                   #S120_SHUTTLE_TO_EXT_LOAD_UNLOAD_POS_START_REQ:
                       REGION S120_SHUTTLE_TO_EXT_LOAD_UNLOAD_POS_START_REQ
                           IF #sInterface.SequenceReleased AND #sStepForward AND (#iShuttleMoving OR #iShuttleModeSemiAutoPos) THEN
                               #sCurrent_Step_NB := #S130_SHUTTLE_TO_EXT_LOAD_UNLOAD_POS_REACHED;
                               #sCheck_Step_Condition := FALSE;
                           END_IF;
                       END_REGION
                   #S130_SHUTTLE_TO_EXT_LOAD_UNLOAD_POS_REACHED:
                       REGION S130_SHUTTLE_TO_EXT_LOAD_UNLOAD_POS_REACHED
                           IF #sInterface.SequenceReleased AND #sStepForward AND NOT #sShuttleStartReq AND #iShuttleModeSemiAutoPos THEN
                               #sCurrent_Step_NB := #S140_STOP_CYCLE;
                               #sCheck_Step_Condition := FALSE;
                           END_IF;
                       END_REGION
                   #S140_STOP_CYCLE:
                       REGION S140_STOP_CYCLE
                           IF #sInterface.SequenceReleased AND #sStepForward AND #iNC_Stopped THEN
                               #sCurrent_Step_NB := #S150_WAIT_OPERATOR_RESTART;
                               #sCheck_Step_Condition := FALSE;
                           END_IF;
                       END_REGION
                       #S150_WAIT_OPERATOR_RESTART:
                           REGION S150_EXCHANGE_EXT_LOADER_IN_PROGRESS
                               IF #sInterface.SequenceReleased AND #sStepForward AND #iOperatorCycleRestart THEN
                                   #sCurrent_Step_NB := #S160_NC_RESTART;
                                   #sCheck_Step_Condition := FALSE;
                               END_IF;
                           END_REGION
                       #S160_NC_RESTART:
                           REGION S60_NC_RESTART
                               IF #sInterface.SequenceReleased AND #sStepForward AND #iNC_Running THEN
                                   #sCurrent_Step_NB := #S170_UPDATE_NEXT_STEP;
                                   #sCheck_Step_Condition := FALSE;
                               END_IF;
                           END_REGION
                       #S170_UPDATE_NEXT_STEP:
                           REGION S70_UPDATE_NEXT_STEP
                               IF #sInterface.SequenceReleased AND #sStepForward AND "AlwaysTRUE" THEN
                                   #sCurrent_Step_NB := #S295_JOB_DONE;
                                   #sCheck_Step_Condition := FALSE;
                               END_IF;
                           END_REGION
                       #S270_UPDATE_NEXT_STEP:
                           REGION S270_UPDATE_NEXT_STEP
                               IF #sInterface.SequenceReleased AND #sStepForward AND "AlwaysTRUE" THEN
                                   #sCurrent_Step_NB := #S295_JOB_DONE;
                                   #sCheck_Step_Condition := FALSE;
                               END_IF;
                           END_REGION
                       #S295_JOB_DONE:
                           REGION S295_JOB_DONE
                               IF NOT #iJobReq THEN
                                   #sCurrent_Step_NB := #S00_INIT;
                                   #sCheck_Step_Condition := FALSE;
                                   #sInterface.JobDone := FALSE;
                               END_IF;
                           END_REGION
               ELSE
                   #sInterface.Error := TRUE;
           END_CASE;
       END_IF;
   END_REGION

   REGION Outputs Update
       #oShuttleStartReq := #sShuttleStartReq;
       #oShuttlePosSetPoint := #sShuttlePosSetPoint;
       #oStopNC_Req := #sStopNC_Req;
       #oRestartNC_Req := #sRestartNC_Req;
       #oRestartStep := #sRestartStep;
       #oContinuationStep := #sContinuationStep;
       #oMsgMissingPart := #sMsgMissingPart;
       #oMsgExtraPart := #sMsgExtraPart;
   END_REGION

   REGION Steps - Date and Time History
       IF #sHistory.Activation THEN
           IF #sHistory.Steps[0] <> #sCurrent_Step_NB THEN
               FOR #tIndex := 98 TO 0 BY -1 DO
                   #sHistory.Steps[#tIndex + 1] := #sHistory.Steps[#tIndex];
                   #sHistory.Date_Time[#tIndex + 1] := #sHistory.Date_Time[#tIndex];
               END_FOR;
               #sHistory.Steps[0] := #sCurrent_Step_NB;
               #sHistory.Date_Time[0] := #iPLC_DateAndTime;
           END_IF;
       END_IF;
   END_REGION

   REGION Steps Text
       #StepText(iErrorCode := #sCurrent_Step_NB,
                 oErrorText => #StepText.oErrorText);
   END_REGION
END_FUNCTION_BLOCK

FUNCTION_BLOCK "FB_LoaderShuttle2"   // FB205, SCL
{ S7_Optimized_Access := 'TRUE' }
// stored: AutoNumber false, MemoryReserve 100, SetENOAutomatically false
   VAR_INPUT
      iGripperReserved : Bool;
      iGripperReleased : Bool;
      iShuttleMoving : Bool;
      iShuttleInPos : Bool;
      iAxisV_Moving : Bool;
      iAxisV_InPos : Bool;
      iAxisW_Moving : Bool;
      iAxisW_InPos : Bool;
   END_VAR
   VAR_OUTPUT
      oExtGateOpenReq : Bool;
      oExtGateCloseReq : Bool;
      oIntGateOpenReq : Bool;
      oIntGateCloseReq : Bool;
      oLoadGripperCloseReq : Bool;
      oUnloadGripperOpenReq : Bool;
      oBlowingReq : Bool;
      oShuttleStartReq : Bool;
      oShuttlePosSetPoint : Real;
      oAxisVStartReq : Bool;
      oAxisVPosSetPoint : Real;
      oAxisWStartReq : Bool;
      oAxisWPosSetPoint : Real;
   END_VAR
   VAR
      sMain : "FB_Main";
      sShuttleInt { S7_SetPoint := 'True'} : "FB_ShuttleInt";
      sShuttleExt { S7_SetPoint := 'True'} : "FB_ShuttleExt";
      sControlIn { S7_SetPoint := 'True'} : "FB_PartControl";
      sControlOut { S7_SetPoint := 'True'} : "FB_PartControl";
      sBlowing { S7_SetPoint := 'True'} : "FB_Blowing";
      sIntLoadUnload { S7_SetPoint := 'True'} : "FB_IntLoadUnload";
      sExtLoadUnload { S7_SetPoint := 'True'} : "FB_ExtLoadUnload";
      sBwLoadUnload { S7_SetPoint := 'True'} : "FB_BwLoadUnload";
      sBwControlIn { S7_SetPoint := 'True'} : "FB_BwControl";
      sActPartControlIn { S7_SetPoint := 'True'} : "FB_ActControl";
      sActPartControlout { S7_SetPoint := 'True'} : "FB_ActControl";
      sActBwControlIn { S7_SetPoint := 'True'} : "FB_ActControl";
      sIntLoadUnloadOP { S7_SetPoint := 'True'} : "FB_IntLoadUnloadOP";
      sBwConsecutiveCtrl_1 { S7_SetPoint := 'True'} : "FB_Consecutive";
      sBwConsecutiveCtrl { S7_SetPoint := 'True'} : "FB_Consecutive";
      sShuttlePosInt { S7_SetPoint := 'True'} : Bool;
      sShuttlePosSas : Bool;
      sShuttlePosExt : Bool;
      sGripper_OK : Bool;
      sExtLoaderInSafePos : Bool;
      sIntLoaderInSafePos : Bool;
      sBwLoaderInSafePos : Bool;
      sRT_PartControlInMissing : R_TRIG;
      sRT_PartControlInExtra : R_TRIG;
      sRT_PartControlOutMissing : R_TRIG;
      sRT_PartControlOutExtra : R_TRIG;
      sRT_BwControlInMissing : R_TRIG;
      sRT_BwControlInExtra : R_TRIG;
      sStepPauseSeq { S7_SetPoint := 'True'} : Bool;
   END_VAR
   VAR_TEMP
      tAxis_U_Position : Struct
         ExtLoadUnloadAuto : Bool;
         ExtLoadUnloadManu : Bool;
         PartControl : Bool;
         BwLoad : Bool;
         BwUnload : Bool;
         BwControl : Bool;
         IntLoadUnload : Bool;
         Blowing : Bool;
         IntLoadUnloadOP : Bool;
      END_STRUCT;
      tAxis_V_Position : Struct
         LoadUnload : Bool;
         Safe : Bool;
         Blowing : Bool;
      END_STRUCT;
      tAxis_W_Position : Struct
         LoadUnload : Bool;
         Safe : Bool;
         Approach : Bool;
         Blowing : Bool;
      END_STRUCT;
   END_VAR
BEGIN
   REGION Shuttle 2 position
       // Init Position
       #sShuttlePosInt := FALSE;
       #sShuttlePosSas := FALSE;
       #sShuttlePosExt := FALSE;

       // Check Shuttle (U2 Axis) position
       IF "DB_AxisPosition".sAxis06_U2."$AA_IM" < "DB_AxisPosMachinePLC".Axis_U2.IntGateExt THEN
           #sShuttlePosExt := TRUE;
       ELSIF "DB_AxisPosition".sAxis06_U2."$AA_IM" > "DB_AxisPosMachinePLC".Axis_U2.ExtGateInt THEN
           #sShuttlePosInt := TRUE;
       ELSE
           #sShuttlePosSas := TRUE;
       END_IF;
   END_REGION

   REGION Position Check
       REGION Axis U2
           // Position : External Load / Unload Auto
           "FC_PositionCheck"(iAxisCurrentPos := "DB_AxisPosition".sAxis06_U2."$AA_IM",
                              iAxisTargetPos := "DB_AxisPosMachinePLC".Axis_U2.ExtLoadUnloadAuto,
                              iTolMin := 0.001,
                              iTolMax := 0.001,
                              iInPos => #tAxis_U_Position.ExtLoadUnloadAuto);

           // Position : External Load / Unload Manu
           "FC_PositionCheck"(iAxisCurrentPos := "DB_AxisPosition".sAxis06_U2."$AA_IM",
                              iAxisTargetPos := "DB_AxisPosMachinePLC".Axis_U2.ExtLoadUnloadManu,
                              iTolMin := 0.001,
                              iTolMax := 0.001,
                              iInPos => #tAxis_U_Position.ExtLoadUnloadManu);

           // Position : Part Control
           "FC_PositionCheck"(iAxisCurrentPos := "DB_AxisPosition".sAxis06_U2."$AA_IM",
                              iAxisTargetPos := "DB_AxisPosMachinePLC".Axis_U2.PartControl,
                              iTolMin := 0.001,
                              iTolMax := 0.001,
                              iInPos => #tAxis_U_Position.PartControl);

           // Position : Backwall Load
           "FC_PositionCheck"(iAxisCurrentPos := "DB_AxisPosition".sAxis06_U2."$AA_IM",
                              iAxisTargetPos := "DB_AxisPosMachinePLC".Axis_U2.BwLoad,
                              iTolMin := 0.001,
                              iTolMax := 0.001,
                              iInPos => #tAxis_U_Position.BwLoad);

           // Position : Backwall Unload
           "FC_PositionCheck"(iAxisCurrentPos := "DB_AxisPosition".sAxis06_U2."$AA_IM",
                              iAxisTargetPos := "DB_AxisPosMachinePLC".Axis_U2.BwUnLoad,
                              iTolMin := 0.001,
                              iTolMax := 0.001,
                              iInPos => #tAxis_U_Position.BwUnload);

           // Position : Backwall Control
           "FC_PositionCheck"(iAxisCurrentPos := "DB_AxisPosition".sAxis06_U2."$AA_IM",
                              iAxisTargetPos := "DB_AxisPosMachinePLC".Axis_U2.BwControl,
                              iTolMin := 0.001,
                              iTolMax := 0.001,
                              iInPos => #tAxis_U_Position.BwControl);

           // Position : Internal Load / Unload
           "FC_PositionCheck"(iAxisCurrentPos := "DB_AxisPosition".sAxis06_U2."$AA_IM",
                              iAxisTargetPos := "DB_AxisPosMachinePLC".Axis_U2.IntLoadUnload,
                              iTolMin := 0.001,
                              iTolMax := 0.001,
                              iInPos => #tAxis_U_Position.IntLoadUnload);

           // Position : Internal Load / Unload OP
           "FC_PositionCheck"(iAxisCurrentPos := "DB_AxisPosition".sAxis06_U2."$AA_IM",
                              iAxisTargetPos := "DB_AxisPosMachinePLC".Axis_U2.IntLoadUnloadOP,
                              iTolMin := 0.001,
                              iTolMax := 0.001,
                              iInPos => #tAxis_U_Position.IntLoadUnloadOP);

           // Position : Blowing (Undrilled part)
           "FC_PositionCheck"(iAxisCurrentPos := "DB_AxisPosition".sAxis06_U2."$AA_IM",
                              iAxisTargetPos := "DB_AxisPosMachinePLC".Axis_U2.Blowing,
                              iTolMin := 0.001,
                              iTolMax := 0.001,
                              iInPos => #tAxis_U_Position.Blowing);
       END_REGION

       REGION Axis V
           // Position : Load / Unload Auto
           "FC_PositionCheck"(iAxisCurrentPos := "DB_AxisPosition".sAxis07_V."$AA_IM",
                              iAxisTargetPos := "DB_AxisPosMachinePLC".Axis_V.Shuttle_2.LoadUnload,
                              iTolMin := 0.001,
                              iTolMax := 0.001,
                              iInPos => #tAxis_V_Position.LoadUnload);

           // Position : Safe
           "FC_PositionCheck"(iAxisCurrentPos := "DB_AxisPosition".sAxis07_V."$AA_IM",
                              iAxisTargetPos := "DB_AxisPosMachinePLC".Axis_V.Safe,
                              iTolMin := 0.001,
                              iTolMax := 0.001,
                              iInPos => #tAxis_V_Position.Safe);

           // Position : Blowing
           "FC_PositionCheck"(iAxisCurrentPos := "DB_AxisPosition".sAxis07_V."$AA_IM",
                              iAxisTargetPos := "DB_AxisPosMachinePLC".Axis_V.Shuttle_2.Blowing,
                              iTolMin := 0.001,
                              iTolMax := 0.001,
                              iInPos => #tAxis_V_Position.Blowing);
       END_REGION

       REGION Axis W
           // Position : Load / Unload Auto
           "FC_PositionCheck"(iAxisCurrentPos := "DB_AxisPosition".sAxis08_W."$AA_IM",
                              iAxisTargetPos := "DB_AxisPosMachinePLC".Axis_W.Shuttle_2.LoadUnload,
                              iTolMin := 0.001,
                              iTolMax := 0.001,
                              iInPos => #tAxis_W_Position.LoadUnload);

           // Position : Safe
           "FC_PositionCheck"(iAxisCurrentPos := "DB_AxisPosition".sAxis08_W."$AA_IM",
                              iAxisTargetPos := "DB_AxisPosMachinePLC".Axis_W.Safe,
                              iTolMin := 0.001,
                              iTolMax := 0.001,
                              iInPos => #tAxis_W_Position.Safe);

           // Position : Approach (confondu avec load/unload)
           "FC_PositionCheck"(iAxisCurrentPos := "DB_AxisPosition".sAxis08_W."$AA_IM",
                              iAxisTargetPos := "DB_AxisPosMachinePLC".Axis_W.Shuttle_2.Approach,
                              iTolMin := 0.001,
                              iTolMax := 0.001,
                              iInPos => #tAxis_W_Position.Approach);

           // Position : Blowing
           "FC_PositionCheck"(iAxisCurrentPos := "DB_AxisPosition".sAxis08_W."$AA_IM",
                              iAxisTargetPos := "DB_AxisPosMachinePLC".Axis_W.Shuttle_2.Blowing,
                              iTolMin := 0.001,
                              iTolMax := 0.001,
                              iInPos => #tAxis_W_Position.Blowing);
       END_REGION
   END_REGION

   REGION Step Pause Sequence
       #sStepPauseSeq := "LBP_ModeGroup".E_JOG
       OR "DB_CycleStartStop".sResquestStopNextCycle
       OR "LBP_Chan1".E_M01;

       #sMain.iStepPause := #sStepPauseSeq;
       #sShuttleInt.iStepPause := #sStepPauseSeq;
       #sShuttleExt.iStepPause := #sStepPauseSeq;
       #sIntLoadUnload.iStepPause := #sStepPauseSeq;
       #sIntLoadUnloadOP.iStepPause := #sStepPauseSeq;
       #sControlIn.iStepPause := #sStepPauseSeq;
       #sControlOut.iStepPause := #sStepPauseSeq;
       #sBwLoadUnload.iStepPause := #sStepPauseSeq;
       #sBwControlIn.iStepPause := #sStepPauseSeq;
       #sBlowing.iStepPause := #sStepPauseSeq;
       #sActPartControlIn.iStepPause := FALSE;
       #sActPartControlout.iStepPause := FALSE;
       #sActBwControlIn.iStepPause := FALSE;
   END_REGION

   REGION Main
       // Gripper prêt à Charger / Décharger une pièce
       #sGripper_OK :=
       ((("DB_PartManagement".sPosition.sShuttle2.Undrilled.Presence.Part AND NOT "DB_PartManagement".sPosition.sGripper.Undrilled.Presence.Part AND "DB_GestionGripper".sUndrilledGripper.oStateOpen) OR NOT "DB_PartManagement".sPosition.sShuttle2.Undrilled.Presence.Part)
       AND (("DB_PartManagement".sPosition.sGripper.Drilled.Presence.Part AND NOT "DB_PartManagement".sPosition.sShuttle2.Drilled.Presence.Part) OR NOT "DB_PartManagement".sPosition.sGripper.Drilled.Presence.Part));

       // Loader INT in Safe Position
       #sIntLoaderInSafePos := "DB_AxisPosition".sAxis07_V."$AA_IM" >= "DB_AxisPosMachinePLC".Axis_V.Safe
       OR ("DB_AxisPosition".sAxis07_V."$AA_IM" < "DB_AxisPosMachinePLC".Axis_V.Safe AND "DB_AxisPosition".sAxis08_W."$AA_IM" >= "DB_AxisPosMachinePLC".Axis_W.Safe);

       // Loader EXT in Safe Position
       #sExtLoaderInSafePos := "DB_SonplasMain".sSonplasLoader.iOperateInOutCollision;

       // BW Loader in Safe Position
       #sBwLoaderInSafePos := "DB_BwLoaderExchange".Inputs.BwLoaderInSafePos;

       // Test Stop after Emptying with only one Shuttle
       IF ("DB_WorkingModes".sEmptying
           AND NOT "DB_LoaderShuttle1".sMain.iJobReq
           AND "DB_PartManagement".sPosition.sPartNumber.Total <= 1) THEN
           #sMain.iJobReq := FALSE;
       END_IF;
       // Test Stop after Emptying with two Shuttle
       IF ("DB_WorkingModes".sEmptying
           AND "DB_LoaderShuttle1".sMain.iJobReq
           AND #sMain.sCurrent_Step_NB = 122
           AND "DB_PartManagement".sPosition.sPartNumber.Total <= 2) THEN
           #sMain.iJobReq := FALSE;
       END_IF;

       #sMain(iStartSeqCond := "DB_PowerOn".sMachineReadySoft AND NOT "MCP1_In".reset,
              iJobReq := #sMain.iJobReq,      
              iShuttleINT := #sShuttlePosInt,
              iShuttleSAS:= #sShuttlePosSas,
              iShuttleEXT := #sShuttlePosExt,
              iGripperReserved := #iGripperReserved,
              iGripperReleased := #iGripperReleased,
              iShuttleUndrilledPart:= "DB_PartManagement".sPosition.sShuttle2.Undrilled.Presence.Part,
              iShuttleDrilledPart:= "DB_PartManagement".sPosition.sShuttle2.Drilled.Presence.Part,
              iShuttleUndrilledBw:= "DB_PartManagement".sPosition.sShuttle2.Undrilled.Presence.BW,
              iShuttleDrilledBw:= "DB_PartManagement".sPosition.sShuttle2.Drilled.Presence.BW,
              iPartCtrlInOK:=#sControlIn.oPartControlOK,
              iPartCtrlInNOK:=#sControlIn.oPartControlNOK,
              iPartCtrlInContinuationStep:=#sActPartControlIn.oContinuationStep,
              iPartCtrlInRestartStep:=#sActPartControlIn.oRestartStep,
              iPartCtrlOutOK:=#sControlOut.oPartControlOK,
              iPartCtrlOutNOK:=#sControlOut.oPartControlNOK,
              iPartCtrlOutContinuationStep:=#sActPartControlout.oContinuationStep,
              iPartCtrlOutRestartStep:=#sActPartControlout.oRestartStep,
              iBwCtrlInOK:=#sBwControlIn.oBwControlOK,
              iBwCtrlInNOK:=#sBwControlIn.oBwControlNOK,
              iBwCtrlInContinuationStep:=#sActBwControlIn.oContinuationStep,
              iBwCtrlInRestartStep:=#sActBwControlIn.oRestartStep,
              iGripperOK:=#sGripper_OK,
              iNC_NoNeedAxis:=NOT "DB_CommPLC_ISO".sAxisManagedByNC,
              iExtLoaderInSafePos:=#sExtLoaderInSafePos,
              iIntLoaderInSafePos:=#sIntLoaderInSafePos,
              iBwLoaderInSafePos:=#sBwLoaderInSafePos,
              iOnePieceMode:="DB_WorkingModes".sOnePiece,
              iPLC_DateAndTime := "DB_ReadDateAndTime".sDateAndTime,
              iStepPause:=#sMain.iStepPause,
              oGripperAxisRequest => #sMain.oGripperAxisRequest,
              oGripperAxisRelease => #sMain.oGripperAxisRelease,
              oNoExtLoad=>#sMain.oNoExtLoad,
              oBwLoadReq=> #sMain.oBwLoadReq,
              oBwUnloadReq=> #sMain.oBwUnloadReq,
              ioShuttleIntSeq := #sShuttleInt.sInterface,
              ioShuttleExtSeq := #sShuttleExt.sInterface,
              ioControlInSeq := #sControlIn.sInterface,
              ioControlOutSeq := #sControlOut.sInterface,
              ioBlowingSeq:=#sBlowing.sInterface,
              ioIntLoadUnloadSeq := #sIntLoadUnload.sInterface,
              ioIntLoadUnloadOP_Seq:=#sIntLoadUnloadOP.sInterface,
              ioExtLoadUnloadSeq := #sExtLoadUnload.sInterface,
              ioBWLoadUnloadSeq := #sBwLoadUnload.sInterface,
              ioBWControlSeq := #sBwControlIn.sInterface,
              ioActPartControlInSeq:= #sActPartControlIn.sInterface,
              ioActPartControlOutSeq:= #sActPartControlout.sInterface,
              ioActBwControlInSeq:= #sActBwControlIn.sInterface);
   END_REGION

   REGION Msg Sequence Fault
       // Msg 700015 Shuttle 2 Sequence Fault
       IF #sMain.sCurrent_Step_NB = 999 THEN
           "LBP_AlarmMsgs".UserA[00].A70UUxx[15] := TRUE;
       END_IF;
   END_REGION

   REGION Shuttle 2 INT
       // Position INT :
       //  If Blowing : Pos. Blowing else Pos. Load/Unload
       IF "DB_LoaderOptions".Blowing.Disabled THEN
           #sShuttleInt.iShuttlePosIntSetPoint := "DB_AxisPosMachinePLC".Axis_U2.IntLoadUnload;
       ELSE
           #sShuttleInt.iShuttlePosIntSetPoint := "DB_AxisPosMachinePLC".Axis_U2.Blowing;
       END_IF;

       #sShuttleInt(iStartSeqCond := (#sMain.iStartSeqCond AND NOT #sShuttleInt.sInterface.Error AND NOT "DB_LoaderShuttle1".sShuttleInt.sInterface.SequenceRun AND #sShuttleInt.sInterface.StartRequest),
                    iJobReq := #sShuttleInt.sInterface.StartRequest,
                    iIntGateOpened := "DB_DigitalInputs".sInternalGateOpened.sSWStatus,
                    iIntGateClosed := "DB_DigitalInputs".sInternalGateLocked.sSWStatus,
                    iExtGateOpened := "DB_DigitalInputs".sExternalGateOpened.sSWStatus,
                    iExtGateClosed := "DB_DigitalInputs".sExternalGateLocked.sSWStatus,
                    iShuttlePosInt := #sShuttlePosInt,
                    iShuttlePosSas := #sShuttlePosSas,
                    iShuttlePosExt := #sShuttlePosExt,
                    iShuttlePosIntSetPoint := #sShuttleInt.iShuttlePosIntSetPoint,
                    iShuttlePosSasSetPoint := "DB_AxisPosMachinePLC".Axis_U2.Sas,
                    iShuttleMoving := #iShuttleMoving,
                    iShuttleInPos := #iShuttleInPos,
                    iIntLoaderInSafePos := #sIntLoaderInSafePos,
                    iPLC_DateAndTime:= "DB_ReadDateAndTime".sDateAndTime,
                    iStepPause:=#sShuttleInt.iStepPause,      
                    oExtGateOpenReq => #sShuttleInt.oExtGateOpenReq,
                    oExtGateCloseReq => #sShuttleInt.oExtGateCloseReq,
                    oIntGateOpenReq => #sShuttleInt.oIntGateOpenReq,
                    oIntGateCloseReq => #sShuttleInt.oIntGateCloseReq,
                    oShuttleStartReq => #sShuttleInt.oShuttleStartReq,
                    oShuttlePosSetPoint => #sShuttleInt.oShuttlePosSetPoint);
   END_REGION

   REGION Shuttle 2 EXT
       #sShuttleExt(iStartSeqCond := (#sIntLoaderInSafePos AND #sBwLoaderInSafePos AND #sMain.iStartSeqCond AND NOT #sShuttleExt.sInterface.Error AND NOT "DB_LoaderShuttle1".sShuttleExt.sInterface.SequenceRun AND #sShuttleExt.sInterface.StartRequest),
                    iJobReq := #sShuttleExt.sInterface.StartRequest,
                    iIntGateOpened := "DB_DigitalInputs".sInternalGateOpened.sSWStatus,
                    iIntGateClosed := "DB_DigitalInputs".sInternalGateLocked.sSWStatus,
                    iExtGateOpened := "DB_DigitalInputs".sExternalGateOpened.sSWStatus,
                    iExtGateClosed := "DB_DigitalInputs".sExternalGateLocked.sSWStatus,
                    iShuttlePosInt := #sShuttlePosInt,
                    iShuttlePosSas := #sShuttlePosSas,
                    iShuttlePosExt := #sShuttlePosExt,
                    iShuttlePosExtSetPoint := "DB_AxisPosMachinePLC".Axis_U2.BwUnLoad,
                    iShuttlePosSasSetPoint := "DB_AxisPosMachinePLC".Axis_U2.Sas,
                    iShuttleMoving := #iShuttleMoving,
                    iShuttleInPos := #iShuttleInPos,
                    iExtLoaderInSafePos := #sExtLoaderInSafePos,
                    iPLC_DateAndTime := "DB_ReadDateAndTime".sDateAndTime,
                    iStepPause:=#sShuttleExt.iStepPause,      
                    oExtGateOpenReq => #sShuttleExt.oExtGateOpenReq,
                    oExtGateCloseReq => #sShuttleExt.oExtGateCloseReq,
                    oIntGateOpenReq => #sShuttleExt.oIntGateOpenReq,
                    oIntGateCloseReq => #sShuttleExt.oIntGateCloseReq,
                    oShuttleStartReq => #sShuttleExt.oShuttleStartReq,
                    oShuttlePosSetPoint => #sShuttleExt.oShuttlePosSetPoint);
   END_REGION

   REGION Ext_LoadUnload
       #sExtLoadUnload(iStartSeqCond := (#sExtLoaderInSafePos AND #sMain.iStartSeqCond AND NOT #sExtLoadUnload.sInterface.Error AND NOT "DB_LoaderShuttle1".sExtLoadUnload.sInterface.SequenceRun AND #sExtLoadUnload.sInterface.StartRequest AND #sShuttlePosExt),
                       iJobReq := #sExtLoadUnload.sInterface.StartRequest,
                       iShuttleExtLoadUnloadAutoPos := #tAxis_U_Position.ExtLoadUnloadAuto,
                       iShuttleExtLoadUnloadAutoPosSetPoint := "DB_AxisPosMachinePLC".Axis_U2.ExtLoadUnloadAuto,
                       iShuttleExtLoadUnloadManuPos := #tAxis_U_Position.ExtLoadUnloadManu,
                       iShuttleExtLoadUnloadManuPosSetPoint := "DB_AxisPosMachinePLC".Axis_U2.ExtLoadUnloadManu,
                       iShuttleMoving := #iShuttleMoving,
                       iShuttleInPos := #iShuttleInPos,
                       iCommunicationWithExtLoaderDone := "DB_SonplasMain".sSonplasLoader.iPartInShuttle2Finished,
                       iLoadUnloadMsgManuModeAck := #sExtLoadUnload.iLoadUnloadMsgManuModeAck OR "MCP1_In".plus OR "DI_SemiAutoValid", // WFA TBD
                       iAutoMode := "DB_WorkingModes".sAuto,
                       iSemiAutoMode := "DB_WorkingModes".sSemiAuto,
                       iFillingMode := "DB_WorkingModes".sFilling AND NOT #sMain.oNoExtLoad,
                       iEmptyingMode := "DB_WorkingModes".sEmptying OR #sMain.oNoExtLoad,
                       iPLC_DateAndTime:= "DB_ReadDateAndTime".sDateAndTime,
                       iStepPause:=#sExtLoadUnload.iStepPause,      
                       oShuttleStartReq => #sExtLoadUnload.oShuttleStartReq,
                       oShuttlePosSetPoint => #sExtLoadUnload.oShuttlePosSetPoint,
                       oStartCommunicationWithExtLoader => "DB_SonplasMain".sSonplasLoader.oPartOutShuttle2InPos,
                       oSetLoadUnloadMsgManuMode => #sExtLoadUnload.oSetLoadUnloadMsgManuMode);

       // Message "Part loaded by operator"
       // IF #sExtLoadUnload.oSetLoadUnloadMsgManuMode THEN
       //     "LBP_AlarmMsgs".UserA[00].A70UUxx[55] := TRUE;
       // ELSIF
       //     #sExtLoadUnload.iLoadUnloadMsgManuModeAck OR "LBP_Chan1".A_Reset THEN
       //     "LBP_AlarmMsgs".UserA[00].A70UUxx[55] := FALSE;
       // END_IF;
       "LBP_AlarmMsgs".UserA[00].A70UUxx[55] := FALSE;
        #sExtLoadUnload.iLoadUnloadMsgManuModeAck := FALSE;
   END_REGION

   REGION Int_LoadUnload
       // Load Gripper Closed according to dry run working mode
        #sIntLoadUnload.iLoadGripperClosed := ("DB_GestionGripper".sUndrilledGripper.oStateCloseWithPart AND NOT "DB_WorkingModes".sDryRun) 
       OR ("DB_GestionGripper".sUndrilledGripper.oStateClose AND "DB_WorkingModes".sDryRun);

       #sIntLoadUnload(iStartSeqCond := (#sIntLoaderInSafePos AND #sMain.iStartSeqCond AND NOT #sIntLoadUnload.sInterface.Error AND NOT "DB_LoaderShuttle1".sIntLoadUnload.sInterface.SequenceRun AND #sIntLoadUnload.sInterface.StartRequest AND #sShuttlePosInt),
                       iJobReq := #sIntLoadUnload.sInterface.StartRequest,
                       iShuttleIntLoadUnloadPos := #tAxis_U_Position.IntLoadUnload,
                       iShuttleIntLoadUnloadPosSetPoint := "DB_AxisPosMachinePLC".Axis_U2.IntLoadUnload,
                       iAxisV_LoadUnloadShuttlePos := #tAxis_V_Position.LoadUnload,
                       iAxisV_LoadUnloadShuttlePosSetPoint := "DB_AxisPosMachinePLC".Axis_V.Shuttle_2.LoadUnload,
                       iAxisV_SafePos := #tAxis_V_Position.Safe,
                       iAxisV_SafePosSetPoint := "DB_AxisPosMachinePLC".Axis_V.Safe,
                       iAxisW_SafePos := #tAxis_W_Position.Safe,
                       iAxisW_SafePosSetPoint := "DB_AxisPosMachinePLC".Axis_W.Safe,
                       iAxisW_ApproachLoadUnloadPos := #tAxis_W_Position.Approach,
                       iAxisW_ApproachLoadUnloadSetPoint := "DB_AxisPosMachinePLC".Axis_W.Shuttle_2.Approach,
                       iAxisW_LoadUnloadPos := #tAxis_W_Position.LoadUnload,
                       iAxisW_LoadUnloadPosSetPoint := "DB_AxisPosMachinePLC".Axis_W.Shuttle_2.LoadUnload,
                       iShuttleMoving := #iShuttleMoving,
                       iShuttleInPos := #iShuttleInPos,
                       iAxisV_Moving := #iAxisV_Moving,
                       iAxisW_InPos := #iAxisW_InPos,
                       iAxisV_InPos := #iAxisV_InPos,
                       iAxisW_Moving := #iAxisW_Moving,
                       iDrilledPartToUnload:= "DB_PartManagement".sPosition.sGripper.Drilled.Presence.Part,
                       iUnDrilledPartToLoad:= "DB_PartManagement".sPosition.sShuttle2.Undrilled.Presence.Part,
                       iLoadGripperClosed := #sIntLoadUnload.iLoadGripperClosed,
                       iUnloadGripperOpen := "DB_GestionGripper".sDrilledGripper.oStateOpen,
                       iPLC_DateAndTime:= "DB_ReadDateAndTime".sDateAndTime,
                       iStepPause:=#sIntLoadUnload.iStepPause,      
                       oShuttleStartReq => #sIntLoadUnload.oShuttleStartReq,
                       oShuttlePosSetPoint => #sIntLoadUnload.oShuttlePosSetPoint,
                       oAxisV_StartReq => #sIntLoadUnload.oAxisV_StartReq,
                       oAxisV_PosSetPoint => #sIntLoadUnload.oAxisV_PosSetPoint,
                       oAxisW_StartReq => #sIntLoadUnload.oAxisW_StartReq,
                       oAxisW_PosSetPoint => #sIntLoadUnload.oAxisW_PosSetPoint,
                       oLoadGripperCloseReq => #sIntLoadUnload.oLoadGripperCloseReq,
                       oUnloadGripperOpenReq => #sIntLoadUnload.oUnloadGripperOpenReq);
   END_REGION

   REGION Int_LoadUnloadOP
           // Load Gripper Closed according to dry run working mode
            #sIntLoadUnloadOP.iLoadGripperClosed := ("DB_GestionGripper".sUndrilledGripper.oStateCloseWithPart AND NOT "DB_WorkingModes".sDryRun) // WFA A Remettre
            OR ("DB_GestionGripper".sUndrilledGripper.oStateClose AND "DB_WorkingModes".sDryRun);

    #sIntLoadUnloadOP(iStartSeqCond := (#sIntLoaderInSafePos AND #sMain.iStartSeqCond AND NOT #sIntLoadUnloadOP.sInterface.Error AND NOT "DB_LoaderShuttle1".sIntLoadUnloadOP.sInterface.SequenceRun AND #sIntLoadUnloadOP.sInterface.StartRequest AND #sShuttlePosInt),
                      iJobReq := #sIntLoadUnloadOP.sInterface.StartRequest,
                      iShuttleIntLoadUnloadPos := #tAxis_U_Position.IntLoadUnload,
                      iShuttleIntLoadUnloadPosSetPoint := "DB_AxisPosMachinePLC".Axis_U2.IntLoadUnload,
                      iShuttleIntLoadUnloadOP_Pos:=#tAxis_U_Position.IntLoadUnloadOP,
                      iShuttleIntLoadUnloadOP_PosSetPoint:="DB_AxisPosMachinePLC".Axis_U2.IntLoadUnloadOP,
                      iAxisV_LoadUnloadShuttlePos := #tAxis_V_Position.LoadUnload,
                      iAxisV_LoadUnloadShuttlePosSetPoint := "DB_AxisPosMachinePLC".Axis_V.Shuttle_2.LoadUnload,
                      iAxisV_SafePos := #tAxis_V_Position.Safe,
                      iAxisV_SafePosSetPoint := "DB_AxisPosMachinePLC".Axis_V.Safe,
                      iAxisW_SafePos := #tAxis_W_Position.Safe,
                      iAxisW_SafePosSetPoint := "DB_AxisPosMachinePLC".Axis_W.Safe,
                      iAxisW_ApproachLoadUnloadPos := #tAxis_W_Position.Approach,
                      iAxisW_ApproachLoadUnloadSetPoint := "DB_AxisPosMachinePLC".Axis_W.Shuttle_2.Approach,
                      iAxisW_LoadUnloadPos := #tAxis_W_Position.LoadUnload,
                      iAxisW_LoadUnloadPosSetPoint := "DB_AxisPosMachinePLC".Axis_W.Shuttle_2.LoadUnload,
                      iShuttleMoving := #iShuttleMoving,
                      iShuttleInPos := #iShuttleInPos,
                      iAxisV_Moving := #iAxisV_Moving,
                      iAxisW_InPos := #iAxisW_InPos,
                      iAxisV_InPos := #iAxisV_InPos,
                      iAxisW_Moving := #iAxisW_Moving,
                      iDrilledPartToUnload := "DB_PartManagement".sPosition.sGripper.Drilled.Presence.Part,
                      iUnDrilledPartToLoad := "DB_PartManagement".sPosition.sShuttle2.Undrilled.Presence.Part,
                      iLoadGripperClosed := #sIntLoadUnloadOP.iLoadGripperClosed,
                      iUnloadGripperOpen := "DB_GestionGripper".sDrilledGripper.oStateOpen,
                      iPLC_DateAndTime := "DB_ReadDateAndTime".sDateAndTime,
                      iStepPause := #sIntLoadUnloadOP.iStepPause,        
                      oShuttleStartReq => #sIntLoadUnloadOP.oShuttleStartReq,
                      oShuttlePosSetPoint => #sIntLoadUnloadOP.oShuttlePosSetPoint,
                      oAxisV_StartReq => #sIntLoadUnloadOP.oAxisV_StartReq,
                      oAxisV_PosSetPoint => #sIntLoadUnloadOP.oAxisV_PosSetPoint,
                      oAxisW_StartReq => #sIntLoadUnloadOP.oAxisW_StartReq,
                      oAxisW_PosSetPoint => #sIntLoadUnloadOP.oAxisW_PosSetPoint,
                      oLoadGripperCloseReq => #sIntLoadUnloadOP.oLoadGripperCloseReq,
                      oUnloadGripperOpenReq => #sIntLoadUnloadOP.oUnloadGripperOpenReq);
   END_REGION

   REGION Parts Control
       // Control In

       // Expected control result
       IF "DB_WorkingModes".sFilling THEN
           #sControlIn.iExpectedCtrlUndrilled := TRUE;
           #sControlIn.iExpectedCtrlDrilled := FALSE;
       ELSIF "DB_WorkingModes".sNormal THEN
           #sControlIn.iExpectedCtrlUndrilled := TRUE;
           #sControlIn.iExpectedCtrlDrilled := FALSE;
       ELSIF "DB_WorkingModes".sEmptying THEN
           #sControlIn.iExpectedCtrlUndrilled := FALSE;
           #sControlIn.iExpectedCtrlDrilled := FALSE;
       END_IF;

       #sControlIn(iStartSeqCond := (#sExtLoaderInSafePos AND #sMain.iStartSeqCond AND NOT #sControlIn.sInterface.Error AND NOT "DB_LoaderShuttle1".sControlIn.sInterface.SequenceRun AND #sControlIn.sInterface.StartRequest AND #sShuttlePosExt),
                   iJobReq := #sControlIn.sInterface.StartRequest,
                   iCtrlEnabled := TRUE,
                   iShuttleCtrlPos := #tAxis_U_Position.PartControl,
                   iShuttleCtrlPosSetPoint := "DB_AxisPosMachinePLC".Axis_U2.PartControl,
                   iExpectedCtrlUndrilled := #sControlIn.iExpectedCtrlUndrilled,
                   iExpectedCtrlDrilled := #sControlIn.iExpectedCtrlDrilled,
                   iUndrilledPartPresence:= "DB_DigitalInputsBW_Station".sUndrilledPartCtrl.sSWStatus,
                   iDrilledPartPresence:= "DB_DigitalInputsBW_Station".sDrilledPartCtrl.sSWStatus,
                   iShuttleMoving := #iShuttleMoving,
                   iShuttleInPos := #iShuttleInPos,
                   iPLC_DateAndTime := "DB_ReadDateAndTime".sDateAndTime,
                   iStepPause := #sControlIn.iStepPause,       
                   oShuttleStartReq => #sControlIn.oShuttleStartReq,
                   oShuttlePosSetPoint => #sControlIn.oShuttlePosSetPoint,
                   oPartControlOK => #sControlIn.oPartControlOK,
                   oPartControlNOK => #sControlIn.oPartControlNOK);

       // Control Out

       // Expected control result
       #sControlOut.iExpectedCtrlUndrilled := "DB_PartManagement".sPosition.sShuttle2.Undrilled.Presence.Part;
       #sControlOut.iExpectedCtrlDrilled := "DB_PartManagement".sPosition.sShuttle2.Drilled.Presence.Part;

       #sControlOut(iStartSeqCond := (#sBwLoaderInSafePos AND #sMain.iStartSeqCond AND NOT #sControlOut.sInterface.Error AND NOT "DB_LoaderShuttle1".sControlOut.sInterface.SequenceRun AND #sControlOut.sInterface.StartRequest AND #sShuttlePosExt),
                    iJobReq := #sControlOut.sInterface.StartRequest,
                    iCtrlEnabled := TRUE,
                    iShuttleCtrlPos := #tAxis_U_Position.PartControl,
                    iShuttleCtrlPosSetPoint := "DB_AxisPosMachinePLC".Axis_U2.PartControl,
                    iExpectedCtrlUndrilled := #sControlOut.iExpectedCtrlUndrilled,
                    iExpectedCtrlDrilled := #sControlOut.iExpectedCtrlDrilled,
                    iUndrilledPartPresence:="DB_DigitalInputsBW_Station".sUndrilledPartCtrl.sSWStatus,
                    iDrilledPartPresence:="DB_DigitalInputsBW_Station".sDrilledPartCtrl.sSWStatus,
                    iShuttleMoving := #iShuttleMoving,
                    iShuttleInPos := #iShuttleInPos,
                    iPLC_DateAndTime := "DB_ReadDateAndTime".sDateAndTime,
                    iStepPause := #sControlOut.iStepPause,      
                    oShuttleStartReq => #sControlOut.oShuttleStartReq,
                    oShuttlePosSetPoint => #sControlOut.oShuttlePosSetPoint,
                    oPartControlOK => #sControlOut.oPartControlOK,
                    oPartControlNOK => #sControlOut.oPartControlNOK);
   END_REGION

   REGION BW Load Unload
       #sBwLoadUnload(iStartSeqCond := (#sMain.iStartSeqCond AND NOT #sBwLoadUnload.sInterface.Error AND NOT "DB_LoaderShuttle1".sBwLoadUnload.sInterface.SequenceRun AND #sBwLoadUnload.sInterface.StartRequest AND #sShuttlePosExt),
                      iJobReq := #sBwLoadUnload.sInterface.StartRequest,
                      iLoadReq:= #sMain.oBwLoadReq,
                      iUnloadReq:= #sMain.oBwUnloadReq,
                      iShuttleBwUnloadPos := #tAxis_U_Position.BwUnload,
                      iShuttleBwUnloadPosSetPoint := "DB_AxisPosMachinePLC".Axis_U2.BwUnLoad,
                      iShuttleBwLoadPos := #tAxis_U_Position.BwLoad,
                      iShuttleBwLoadPosSetPoint := "DB_AxisPosMachinePLC".Axis_U2.BwLoad,
                      iShuttleMoving := #iShuttleMoving,
                      iShuttleInPos := #iShuttleInPos,
                      iBwLoadDone:= "DB_BwLoader".sBwCommunication.oLoadJobDone,
                      iBwUnloadDone:= "DB_BwLoader".sBwCommunication.oUnloadJobDone,
                      iBwLoaderInSafePos:=#sBwLoaderInSafePos,
                      iPLC_DateAndTime:= "DB_ReadDateAndTime".sDateAndTime,
                      iStepPause:=#sBwLoadUnload.iStepPause,      
                      oShuttleStartReq => #sBwLoadUnload.oShuttleStartReq,
                      oShuttlePosSetPoint => #sBwLoadUnload.oShuttlePosSetPoint,
                      oBwLoadReq=>#sBwLoadUnload.oBwLoadReq,
                      oBwUnloadReq=>#sBwLoadUnload.oBwUnloadReq);
   END_REGION

   REGION BW Control
       // BW Control In

       // Expected control result
       #sBwControlIn.iExpectedCtrl := "DB_PartManagement".sPosition.sShuttle2.Undrilled.Presence.Part;

       #sBwControlIn(iStartSeqCond := (#sMain.iStartSeqCond AND NOT #sBwControlIn.sInterface.Error AND NOT "DB_LoaderShuttle1".sBwControlIn.sInterface.SequenceRun AND #sBwControlIn.sInterface.StartRequest AND #sShuttlePosExt),
                     iJobReq := #sBwControlIn.sInterface.StartRequest,
                     iCtrlEnabled := TRUE,
                     iShuttleCtrlPos := #tAxis_U_Position.BwControl,
                     iShuttleCtrlPosSetPoint := "DB_AxisPosMachinePLC".Axis_U2.BwControl,
                     iExpectedCtrl := #sBwControlIn.iExpectedCtrl,
                     iBwPresence := "DB_DigitalInputsBW_Station".sBwCtrl.sSWStatus,
                     iShuttleMoving := #iShuttleMoving,
                     iShuttleInPos := #iShuttleInPos,
                     iPLC_DateAndTime := "DB_ReadDateAndTime".sDateAndTime,
                     iStepPause := #sBwControlIn.iStepPause,   
                     oShuttleStartReq => #sBwControlIn.oShuttleStartReq,
                     oShuttlePosSetPoint => #sBwControlIn.oShuttlePosSetPoint,
                     oBwControlOK => #sBwControlIn.oBwControlOK,
                     oBwControlNOK => #sBwControlIn.oBwControlNOK);

       #sBwConsecutiveCtrl(iReset := #sBwConsecutiveCtrl.oConsecutiveError AND #sActBwControlIn.sCurrent_Step_NB = 60,
                           iGoodEntry := #sBwControlIn.oBwControlOK,
                           iBadEntry := #sBwControlIn.oBwControlNOK,
                           iPresetValue := 3,
                           oConsecutiveError => #sBwConsecutiveCtrl.oConsecutiveError);
   END_REGION

   REGION Blowing
       #sBlowing(iStartSeqCond := (#sIntLoaderInSafePos AND #sMain.iStartSeqCond AND NOT #sBlowing.sInterface.Error AND NOT "DB_LoaderShuttle1".sBlowing.sInterface.SequenceRun AND #sBlowing.sInterface.StartRequest AND #sShuttlePosInt),
                 iJobReq := #sBlowing.sInterface.StartRequest,
                 iShuttleBlowingPos := #tAxis_U_Position.Blowing,
                 iShuttleBlowingPosSetPoint := "DB_AxisPosMachinePLC".Axis_U2.Blowing,
                 iAxisV_BlowingPos := #tAxis_V_Position.Blowing,
                 iAxisV_BlowingPosSetPoint := "DB_AxisPosMachinePLC".Axis_V.Shuttle_2.Blowing,
                 iAxisW_SafePos := #tAxis_W_Position.Safe,
                 iAxisW_SafePosSetPoint := "DB_AxisPosMachinePLC".Axis_W.Safe,
                 iAxisW_BlowingPos := #tAxis_W_Position.Blowing,
                 iAxisW_BlowingPosSetPoint := "DB_AxisPosMachinePLC".Axis_W.Shuttle_2.Blowing,
                 iShuttleMoving := #iShuttleMoving,
                 iShuttleInPos := #iShuttleInPos,
                 iAxisV_Moving := #iAxisV_Moving,
                 iAxisV_InPos := #iAxisV_InPos,
                 iAxisW_Moving := #iAxisW_Moving,
                 iAxisW_InPos := #iAxisW_InPos,
                 iBlowingTime:=DINT_TO_TIME(REAL_TO_DINT("DB_HMISetting".BlowingSetpoint)),
                 iPLC_DateAndTime := "DB_ReadDateAndTime".sDateAndTime,
                 iStepPause := #sBlowing.iStepPause,
                 oShuttleStartReq => #sBlowing.oShuttleStartReq,
                 oShuttlePosSetPoint => #sBlowing.oShuttlePosSetPoint,
                 oAxisV_StartReq => #sBlowing.oAxisV_StartReq,
                 oAxisV_PosSetPoint => #sBlowing.iAxisV_BlowingPosSetPoint,
                 oAxisW_StartReq => #sBlowing.oAxisW_StartReq,
                 oAxisW_PosSetPoint => #sBlowing.iAxisW_BlowingPosSetPoint,
                 oBlowingReq => #sBlowing.oBlowingReq);
   END_REGION

   REGION Action Part Control In
       // Conditions d'arrêt en Mode Auto
       #sActPartControlIn.iModeAutoPosCondition :=
       ("DB_WorkingModes".sAuto AND (#sControlIn.sMissingPartCtrlUndrilled OR #sControlIn.sMissingPartCtrlDrilled) AND "DB_LoaderOptions".ActPartControlIn.Stop)
       OR ("DB_WorkingModes".sAuto AND (#sControlIn.sExtraPartCtrlUndrilled OR #sControlIn.sExtraPartCtrlDrilled) AND "DB_LoaderOptions".ActPartControlIn.Stop)
       OR ("DB_WorkingModes".sAuto AND (#sControlIn.sExtraPartCtrlUndrilled OR #sControlIn.sExtraPartCtrlDrilled) AND NOT "DB_LoaderOptions".ActPartControlIn.Stop);
       // Conditions d'arrêt en Mode Semi Auto   
       #sActPartControlIn.iModeSemiAutoPosCondition :=
       ("DB_WorkingModes".sSemiAuto AND (#sControlIn.sMissingPartCtrlUndrilled OR #sControlIn.sMissingPartCtrlDrilled) AND "DB_LoaderOptions".ActPartControlIn.Stop)
       OR ("DB_WorkingModes".sSemiAuto AND (#sControlIn.sExtraPartCtrlUndrilled OR #sControlIn.sExtraPartCtrlDrilled) AND "DB_LoaderOptions".ActPartControlIn.Stop)
       OR ("DB_WorkingModes".sSemiAuto AND (#sControlIn.sExtraPartCtrlUndrilled OR #sControlIn.sExtraPartCtrlDrilled) AND NOT "DB_LoaderOptions".ActPartControlIn.Stop);
       // Conditions pas d'arrêt
       #sActPartControlIn.iNoStopCondition :=
       ("DB_WorkingModes".sAuto AND (#sControlIn.sMissingPartCtrlUndrilled OR #sControlIn.sMissingPartCtrlDrilled) AND NOT "DB_LoaderOptions".ActPartControlIn.Stop)
       OR ("DB_WorkingModes".sSemiAuto AND (#sControlIn.sMissingPartCtrlUndrilled OR #sControlIn.sMissingPartCtrlDrilled) AND NOT "DB_LoaderOptions".ActPartControlIn.Stop);

       #sActPartControlIn(iStartSeqCond := (#sMain.iStartSeqCond AND NOT #sActPartControlIn.sInterface.Error AND NOT "DB_LoaderShuttle1".sActPartControlIn.sInterface.SequenceRun AND #sActPartControlIn.sInterface.StartRequest AND #sShuttlePosExt),
                          iJobReq := #sActPartControlIn.sInterface.StartRequest,
                          iShuttleModeAutoPos := #tAxis_U_Position.ExtLoadUnloadAuto,
                          iShuttleModeAutoPosSetPoint := "DB_AxisPosMachinePLC".Axis_U2.ExtLoadUnloadAuto,
                          iShuttleModeSemiAutoPos := #tAxis_U_Position.ExtLoadUnloadManu,
                          iShuttleModeSemiAutoPosSetPoint := "DB_AxisPosMachinePLC".Axis_U2.ExtLoadUnloadManu,
                          iShuttleMoving := #iShuttleMoving,
                          iShuttleInPos := #iShuttleInPos,
                          iModeAutoPosCondition := #sActPartControlIn.iModeAutoPosCondition,
                          iModeSemiAutoPosCondition := #sActPartControlIn.iModeSemiAutoPosCondition,
                          iNoStopCondition := #sActPartControlIn.iNoStopCondition,
                          iOperatorCycleRestart := "LBP_Chan1".E_ProgRunning,
                          iNC_Stopped := NOT "LBP_Chan1".E_ProgRunning,
                          iNC_Running := "LBP_Chan1".E_ProgRunning,
                          iMissingPart:=#sControlIn.sMissingPartCtrlUndrilled OR #sControlIn.sMissingPartCtrlDrilled,
                          iExtraPart:=#sControlIn.sExtraPartCtrlUndrilled OR #sControlIn.sExtraPartCtrlDrilled,
                          iPLC_DateAndTime := "DB_ReadDateAndTime".sDateAndTime,
                          iStepPause := #sActPartControlIn.iStepPause,
                          oShuttleStartReq => #sActPartControlIn.oShuttleStartReq,
                          oShuttlePosSetPoint => #sActPartControlIn.oShuttlePosSetPoint,
                          oStopNC_Req => #sActPartControlIn.oStopNC_Req,       // Implicite par Alarm Message
                          oRestartNC_Req => #sActPartControlIn.oRestartNC_Req, // Implicite par Restart NC
                          oRestartStep => #sActPartControlIn.oRestartStep,
                          oContinuationStep => #sActPartControlIn.oContinuationStep,
                          oMsgMissingPart=>#sActPartControlIn.oMsgMissingPart,
                          oMsgExtraPart=>#sActPartControlIn.oMsgExtraPart);

       #sRT_PartControlInMissing(CLK := #sActPartControlIn.oMsgMissingPart);
       IF #sRT_PartControlInMissing.Q THEN
           "LBP_AlarmMsgs".UserA[03].A70UUxx[21] := TRUE;
       END_IF;

       #sRT_PartControlInExtra(CLK := #sActPartControlIn.oMsgExtraPart);
       IF #sRT_PartControlInExtra.Q THEN
           "LBP_AlarmMsgs".UserA[03].A70UUxx[22] := TRUE;
       END_IF;
   END_REGION

   REGION Action Part Control Out
       // Conditions d'arrêt en Mode Auto
       #sActPartControlout.iModeAutoPosCondition :=
       ("DB_WorkingModes".sAuto AND (#sControlOut.sMissingPartCtrlUndrilled OR #sControlOut.sMissingPartCtrlDrilled) AND "DB_LoaderOptions".ActPartControlOut.Stop)
       OR ("DB_WorkingModes".sAuto AND (#sControlOut.sExtraPartCtrlUndrilled OR #sControlOut.sExtraPartCtrlDrilled) AND "DB_LoaderOptions".ActPartControlOut.Stop)
       OR ("DB_WorkingModes".sAuto AND (#sControlOut.sExtraPartCtrlUndrilled OR #sControlOut.sExtraPartCtrlDrilled) AND NOT "DB_LoaderOptions".ActPartControlOut.Stop);
       // Conditions d'arrêt en Mode Semi Auto 
       #sActPartControlout.iModeSemiAutoPosCondition :=
       ("DB_WorkingModes".sSemiAuto AND (#sControlOut.sMissingPartCtrlUndrilled OR #sControlOut.sMissingPartCtrlDrilled) AND "DB_LoaderOptions".ActPartControlOut.Stop)
       OR ("DB_WorkingModes".sSemiAuto AND (#sControlOut.sExtraPartCtrlUndrilled OR #sControlOut.sExtraPartCtrlDrilled) AND "DB_LoaderOptions".ActPartControlOut.Stop)
       OR ("DB_WorkingModes".sSemiAuto AND (#sControlOut.sExtraPartCtrlUndrilled OR #sControlOut.sExtraPartCtrlDrilled) AND NOT "DB_LoaderOptions".ActPartControlOut.Stop);
       // Conditions pas d'arrêt
       #sActPartControlout.iNoStopCondition :=
       ("DB_WorkingModes".sAuto AND (#sControlOut.sMissingPartCtrlUndrilled OR #sControlOut.sMissingPartCtrlDrilled) AND NOT "DB_LoaderOptions".ActPartControlOut.Stop)
       OR ("DB_WorkingModes".sSemiAuto AND (#sControlOut.sMissingPartCtrlUndrilled OR #sControlOut.sMissingPartCtrlDrilled) AND NOT "DB_LoaderOptions".ActPartControlOut.Stop);

       #sActPartControlout(iStartSeqCond := (#sMain.iStartSeqCond AND NOT #sActPartControlout.sInterface.Error AND NOT "DB_LoaderShuttle1".sActPartControlOut.sInterface.SequenceRun AND #sActPartControlout.sInterface.StartRequest AND #sShuttlePosExt),
                           iJobReq := #sActPartControlout.sInterface.StartRequest,
                           iShuttleModeAutoPos := #tAxis_U_Position.ExtLoadUnloadAuto,
                           iShuttleModeAutoPosSetPoint := "DB_AxisPosMachinePLC".Axis_U2.ExtLoadUnloadAuto,
                           iShuttleModeSemiAutoPos := #tAxis_U_Position.ExtLoadUnloadManu,
                           iShuttleModeSemiAutoPosSetPoint := "DB_AxisPosMachinePLC".Axis_U2.ExtLoadUnloadManu,
                           iShuttleMoving := #iShuttleMoving,
                           iShuttleInPos := #iShuttleInPos,
                           iModeAutoPosCondition := #sActPartControlout.iModeAutoPosCondition,
                           iModeSemiAutoPosCondition := #sActPartControlout.iModeSemiAutoPosCondition,
                           iNoStopCondition := #sActPartControlout.iNoStopCondition,
                           iOperatorCycleRestart := "LBP_Chan1".E_ProgRunning,
                           iNC_Stopped := NOT "LBP_Chan1".E_ProgRunning,
                           iNC_Running := "LBP_Chan1".E_ProgRunning,
                           iMissingPart:=#sControlOut.sMissingPartCtrlUndrilled OR #sControlOut.sMissingPartCtrlDrilled,
                           iExtraPart:=#sControlOut.sExtraPartCtrlUndrilled OR #sControlOut.sExtraPartCtrlDrilled,
                           iPLC_DateAndTime := "DB_ReadDateAndTime".sDateAndTime,
                           iStepPause := #sActPartControlout.iStepPause,
                           oShuttleStartReq => #sActPartControlout.oShuttleStartReq,
                           oShuttlePosSetPoint => #sActPartControlout.oShuttlePosSetPoint,
                           oStopNC_Req => #sActPartControlout.oStopNC_Req,       // Implicite par Alarm Message
                           oRestartNC_Req => #sActPartControlout.oRestartNC_Req, // Implicite par Restart NC
                           oRestartStep => #sActPartControlout.oRestartStep,
                           oContinuationStep => #sActPartControlout.oContinuationStep,
                           oMsgMissingPart=>#sActPartControlout.oMsgMissingPart,
                           oMsgExtraPart=>#sActPartControlout.oMsgExtraPart);

       #sRT_PartControlOutMissing(CLK := #sActPartControlout.oMsgMissingPart);
       IF #sRT_PartControlOutMissing.Q THEN
           "LBP_AlarmMsgs".UserA[03].A70UUxx[23] := TRUE;
       END_IF;

       #sRT_PartControlOutExtra(CLK := #sActPartControlout.oMsgExtraPart);
       IF #sRT_PartControlOutExtra.Q THEN
           "LBP_AlarmMsgs".UserA[03].A70UUxx[24] := TRUE;
       END_IF;
   END_REGION

   REGION Action Bw Control In
       // Conditions d'arrêt en Mode Auto
       #sActBwControlIn.iModeAutoPosCondition :=
       ("DB_WorkingModes".sAuto AND #sBwControlIn.sMissingBwCtrl AND ("DB_LoaderOptions".ActBwControlIn.Stop OR #sBwConsecutiveCtrl.oConsecutiveError))
       OR ("DB_WorkingModes".sAuto AND #sBwControlIn.sExtraBwCtrl AND "DB_LoaderOptions".ActBwControlIn.Stop)
       OR ("DB_WorkingModes".sAuto AND #sBwControlIn.sExtraBwCtrl AND NOT "DB_LoaderOptions".ActBwControlIn.Stop);
       // Conditions d'arrêt en Mode Semi Auto
       #sActBwControlIn.iModeSemiAutoPosCondition :=
       ("DB_WorkingModes".sSemiAuto AND #sBwControlIn.sMissingBwCtrl AND "DB_LoaderOptions".ActBwControlIn.Stop)
       OR ("DB_WorkingModes".sSemiAuto AND #sBwControlIn.sExtraBwCtrl AND "DB_LoaderOptions".ActBwControlIn.Stop)
       OR ("DB_WorkingModes".sSemiAuto AND #sBwControlIn.sExtraBwCtrl AND NOT "DB_LoaderOptions".ActBwControlIn.Stop);
       // Conditions pas d'arrêt
       #sActBwControlIn.iNoStopCondition :=
       ("DB_WorkingModes".sAuto AND #sBwControlIn.sMissingBwCtrl AND (NOT "DB_LoaderOptions".ActBwControlIn.Stop AND NOT #sBwConsecutiveCtrl.oConsecutiveError))
       OR ("DB_WorkingModes".sSemiAuto AND #sBwControlIn.sMissingBwCtrl AND NOT "DB_LoaderOptions".ActBwControlIn.Stop);

       #sActBwControlIn(iStartSeqCond := (#sMain.iStartSeqCond AND NOT #sActBwControlIn.sInterface.Error AND NOT "DB_LoaderShuttle1".sActBwControlIn.sInterface.SequenceRun AND #sActBwControlIn.sInterface.StartRequest AND #sShuttlePosExt),
                        iJobReq := #sActBwControlIn.sInterface.StartRequest,
                        iShuttleModeAutoPos := #tAxis_U_Position.BwLoad,
                        iShuttleModeAutoPosSetPoint := "DB_AxisPosMachinePLC".Axis_U2.BwLoad,
                        iShuttleModeSemiAutoPos := #tAxis_U_Position.BwLoad,
                        iShuttleModeSemiAutoPosSetPoint := "DB_AxisPosMachinePLC".Axis_U2.BwLoad,
                        iShuttleMoving := #iShuttleMoving,
                        iShuttleInPos := #iShuttleInPos,
                        iModeAutoPosCondition := #sActBwControlIn.iModeAutoPosCondition,
                        iModeSemiAutoPosCondition := #sActBwControlIn.iModeSemiAutoPosCondition,
                        iNoStopCondition := #sActBwControlIn.iNoStopCondition,
                        iOperatorCycleRestart := "LBP_Chan1".E_ProgRunning,
                        iNC_Stopped :=  (NOT "LBP_Chan1".E_ProgRunning AND "DB_OPC_Machine".Parameters.ConsecutiveBwIn = 0) OR "DB_OPC_Machine".Parameters.ConsecutiveBwIn > 0,
                        iNC_Running := "LBP_Chan1".E_ProgRunning,
                        iMissingPart:=#sBwControlIn.sMissingBwCtrl,
                        iExtraPart:=#sBwControlIn.sExtraBwCtrl,
                        iPLC_DateAndTime := "DB_ReadDateAndTime".sDateAndTime,
                        iStepPause := #sActBwControlIn.iStepPause, 
                        oShuttleStartReq => #sActBwControlIn.oShuttleStartReq,
                        oShuttlePosSetPoint => #sActBwControlIn.oShuttlePosSetPoint,
                        oStopNC_Req => #sActBwControlIn.oStopNC_Req,       // Implicite par Alarm Message
                        oRestartNC_Req => #sActBwControlIn.oRestartNC_Req, // Implicite par Restart NC
                        oRestartStep => #sActBwControlIn.oRestartStep,
                        oContinuationStep => #sActBwControlIn.oContinuationStep,
                        oMsgMissingPart=>#sActBwControlIn.oMsgMissingPart,
                        oMsgExtraPart=>#sActBwControlIn.oMsgExtraPart);

       IF "DB_OPC_Machine".Parameters.ConsecutiveBwIn = 0 THEN
           #sRT_BwControlInMissing(CLK := #sActBwControlIn.oMsgMissingPart);
           IF #sRT_BwControlInMissing.Q THEN
               "LBP_AlarmMsgs".UserA[03].A70UUxx[25] := TRUE;
           END_IF;

           #sRT_BwControlInExtra(CLK := #sActBwControlIn.iExtraPart);
           IF #sRT_BwControlInExtra.Q THEN
               "LBP_AlarmMsgs".UserA[03].A70UUxx[26] := TRUE;
           END_IF;
       ELSE
           "LBP_AlarmMsgs".UserA[03].A70UUxx[25] := FALSE;
           "LBP_AlarmMsgs".UserA[03].A70UUxx[26] := FALSE;
       END_IF;
   END_REGION

   REGION Axis U-V-W Start Request
       // Axis U - Start Request
       #oShuttleStartReq :=
       #sShuttleInt.oShuttleStartReq
       OR #sShuttleExt.oShuttleStartReq
       OR #sControlIn.oShuttleStartReq
       OR #sControlOut.oShuttleStartReq
       OR #sBlowing.oShuttleStartReq
       OR #sIntLoadUnload.oShuttleStartReq
       OR #sIntLoadUnloadOP.oShuttleStartReq
       OR #sExtLoadUnload.oShuttleStartReq
       OR #sBwLoadUnload.oShuttleStartReq
       OR #sBwControlIn.oShuttleStartReq
       OR #sActPartControlIn.oShuttleStartReq
       OR #sActPartControlout.oShuttleStartReq
       OR #sActBwControlIn.oShuttleStartReq;

       // Axis U - Position Set point according to start request
       IF #sShuttleInt.oShuttleStartReq THEN
           #oShuttlePosSetPoint := #sShuttleInt.oShuttlePosSetPoint;
       ELSIF #sShuttleExt.oShuttleStartReq THEN
           #oShuttlePosSetPoint := #sShuttleExt.oShuttlePosSetPoint;
       ELSIF #sControlIn.oShuttleStartReq THEN
           #oShuttlePosSetPoint := #sControlIn.oShuttlePosSetPoint;
       ELSIF #sControlOut.oShuttleStartReq THEN
           #oShuttlePosSetPoint := #sControlOut.oShuttlePosSetPoint;
       ELSIF #sExtLoadUnload.oShuttleStartReq THEN
           #oShuttlePosSetPoint := #sExtLoadUnload.oShuttlePosSetPoint;
       ELSIF #sIntLoadUnload.oShuttleStartReq THEN
           #oShuttlePosSetPoint := #sIntLoadUnload.oShuttlePosSetPoint;
       ELSIF #sIntLoadUnloadOP.oShuttleStartReq THEN
           #oShuttlePosSetPoint := #sIntLoadUnloadOP.oShuttlePosSetPoint;
       ELSIF #sBwLoadUnload.oShuttleStartReq THEN
           #oShuttlePosSetPoint := #sBwLoadUnload.oShuttlePosSetPoint;
       ELSIF #sBwControlIn.oShuttleStartReq THEN
           #oShuttlePosSetPoint := #sBwControlIn.oShuttlePosSetPoint;
       ELSIF #sActPartControlIn.oShuttleStartReq THEN
           #oShuttlePosSetPoint := #sActPartControlIn.oShuttlePosSetPoint;
       ELSIF #sActPartControlout.oShuttleStartReq THEN
           #oShuttlePosSetPoint := #sActPartControlout.oShuttlePosSetPoint;
       ELSIF #sActBwControlIn.oShuttleStartReq THEN
           #oShuttlePosSetPoint := #sActBwControlIn.oShuttlePosSetPoint;
       ELSIF  #sBlowing.oShuttleStartReq THEN
           #oShuttlePosSetPoint := #sBlowing.oShuttlePosSetPoint;
       ELSE
           #oShuttleStartReq := FALSE;
       END_IF;

       // Axis V - Start Request
       #oAxisVStartReq :=
       #sIntLoadUnload.oAxisV_StartReq
       OR #sIntLoadUnloadOP.oAxisV_StartReq
       OR #sBlowing.oAxisV_StartReq;

       // Axis V - Position Set point  according to start request
       IF #sIntLoadUnload.oAxisV_StartReq THEN
           #oAxisVPosSetPoint := #sIntLoadUnload.oAxisV_PosSetPoint;
       ELSIF #sIntLoadUnloadOP.oAxisV_StartReq THEN
           #oAxisVPosSetPoint := #sIntLoadUnloadOP.oAxisV_PosSetPoint;
       ELSIF #sBlowing.oAxisV_StartReq THEN
           #oAxisVPosSetPoint := #sBlowing.oAxisV_PosSetPoint;
       ELSE
           #oAxisVStartReq := FALSE;
       END_IF;

       // Axis W - Start Request
       #oAxisWStartReq :=
       #sIntLoadUnload.oAxisW_StartReq
       OR #sIntLoadUnloadOP.oAxisW_StartReq
       OR #sBlowing.oAxisW_StartReq;

       // Axis W - Position Set point  according to start request
       IF #sIntLoadUnload.oAxisW_StartReq THEN
           #oAxisWPosSetPoint := #sIntLoadUnload.oAxisW_PosSetPoint;
       ELSIF #sIntLoadUnloadOP.oAxisW_StartReq THEN
           #oAxisWPosSetPoint := #sIntLoadUnloadOP.oAxisW_PosSetPoint;
       ELSIF #sBlowing.oAxisW_StartReq THEN
           #oAxisWPosSetPoint := #sBlowing.oAxisW_PosSetPoint;
       ELSE
           #oAxisWStartReq := FALSE;
       END_IF;
   END_REGION

   REGION Gates Command Request
       // External Gate
       #oExtGateOpenReq := #sShuttleInt.oExtGateOpenReq OR #sShuttleExt.oExtGateOpenReq;
       #oExtGateCloseReq := #sShuttleInt.oExtGateCloseReq OR #sShuttleExt.oExtGateCloseReq;

       // Internal Gate
       #oIntGateOpenReq := #sShuttleInt.oIntGateOpenReq OR #sShuttleExt.oIntGateOpenReq;
       #oIntGateCloseReq := #sShuttleInt.oIntGateCloseReq OR #sShuttleExt.oIntGateCloseReq;
   END_REGION

   REGION Gripper Command Request
       // Load Gripper
       #oLoadGripperCloseReq := #sIntLoadUnload.oLoadGripperCloseReq
       OR #sIntLoadUnloadOP.oLoadGripperCloseReq;
       // Unload Gripper
       #oUnloadGripperOpenReq := #sIntLoadUnload.oUnloadGripperOpenReq
       OR #sIntLoadUnloadOP.oUnloadGripperOpenReq;
   END_REGION

   REGION Blowing Command Request
       #oBlowingReq := #sBlowing.oBlowingReq;
   END_REGION
END_FUNCTION_BLOCK

FUNCTION_BLOCK "FB_LoaderAxis"   // FB206, SCL
{ S7_Optimized_Access := 'TRUE' }
// stored: AutoNumber false, MemoryReserve 100, SetENOAutomatically false
   VAR_INPUT
      iPLCModeReq : Bool;   // Axis Managed by PLC Request
      iCNCModeReq : Bool;   // Axis Managed by CNC Request
      iU1StartReq : Bool;   // Axis U1 Start Request
      iU2StartReq : Bool;   // Axis U2 Start Request
      iVStartReq : Bool;   // Axis V Start Request
      iWStartReq : Bool;   // Axis W Start Request
      iU1PosSetPoint : Real;   // Axis U1 Position Setpoint
      iU2PosSetPoint : Real;   // Axis U2 Position Setpoint
      iVPosSetPoint : Real;   // Axis V Position Setpoint
      iWPosSetPoint : Real;   // Axis W Position Setpoint
   END_VAR
   VAR_OUTPUT
      oU1InPos : Bool;   // Axis U1 Position Reached
      oU2InPos : Bool;   // Axis U2 Position Reached
      oVInPos : Bool;   // Axis V Position Reached
      oWInPos : Bool;   // Axis W Position Reached
   END_VAR
   VAR
      sAxisPLCMode : Bool := false;
      sAxisCNCMode : Bool := false;
      sAllAxisPLCMode : Bool := false;
      sAllAxisCNCMode : Bool := false;
      sU1StartMove : Bool;
      sU2StartMove : Bool;
      sVStartMove : Bool;
      sWStartMove : Bool;
      sU1MoveError : Bool;
      sU2MoveError : Bool;
      sVMoveError : Bool;
      sWMoveError : Bool;
      sU1InPos : Bool;
      sU2InPos : Bool;
      sVInPos : Bool;
      sWInPos : Bool;
      sU1SetPos : Real;
      sU2SetPos : Real;
      sVSetPos : Real;
      sWSetPos : Real;
      sU1MoveState : Byte;
      sU2MoveState : Byte;
      sVMoveState : Byte;
      sWMoveState : Byte;
      sU1ActFeedRate : LReal;
      sU2ActFeedRate : LReal;
      sVActFeedRate : LReal;
      sWActFeedRate : LReal;
      sU1DrivedByPLC : Bool;
      sU2DrivedByPLC : Bool;
      sVDrivedByPLC : Bool;
      sWDrivedByPLC : Bool;
      sU1Positioning { ExternalAccessible := 'False'; ExternalVisible := 'False'; ExternalWritable := 'False'} : Bool;
      sU2Positioning { ExternalAccessible := 'False'; ExternalVisible := 'False'; ExternalWritable := 'False'} : Bool;
      sVPositioning { ExternalAccessible := 'False'; ExternalVisible := 'False'; ExternalWritable := 'False'} : Bool;
      sWPositioning { ExternalAccessible := 'False'; ExternalVisible := 'False'; ExternalWritable := 'False'} : Bool;
      sFeedActive : Bool;
   END_VAR
BEGIN
   REGION Update Inputs
       #sU1StartMove := #iU1StartReq;
       #sU2StartMove := #iU2StartReq;
       #sVStartMove  := #iVStartReq;
       #sWStartMove  := #iWStartReq;

       #sU1SetPos := #iU1PosSetPoint;
       #sU2SetPos := #iU2PosSetPoint;
       #sVSetPos  := #iVPosSetPoint;
       #sWSetPos  := #iWPosSetPoint;
   END_REGION


   REGION Feed Active/Axis moving
       #sU1Positioning := "LBP_Axis05_U1".E_PosAxis AND "LBP_Axis05_U1".E_PLCASp;
       #sU2Positioning := "LBP_Axis06_U2".E_PosAxis AND "LBP_Axis06_U2".E_PLCASp;
       #sVPositioning  := "LBP_Axis07_V".E_PosAxis  AND "LBP_Axis07_V".E_PLCASp;
       #sWPositioning  := "LBP_Axis08_W".E_PosAxis  AND "LBP_Axis08_W".E_PLCASp;

       #sFeedActive := //  A least 1 axis is moving
       ("LBP_Chan1".A_FD_OR <> B#16#1)  // Speed more than 0
       AND (#sU1Positioning             // Axis06 U1 moving
           OR #sU2Positioning           // Axis09 U2 moving
           OR #sVPositioning            // Axis07 V  moving
           OR #sWPositioning);          // Axis08 W  moving
   END_REGION

   REGION Axis CNC mode (Only when NC in JOG Mode)
       IF #sAxisPLCMode
           AND #iCNCModeReq
           OR "MCP1_In".reset
           OR NOT "DB_DataFromSafety".EmergencyStop THEN
           #sAxisCNCMode := TRUE;
           #sAxisPLCMode := FALSE;
       END_IF;

       #sAllAxisCNCMode :=
           NOT "LBP_Axis05_U1".E_PLCASp
       AND NOT "LBP_Axis06_U2".E_PLCASp
       AND NOT "LBP_Axis07_V".E_PLCASp
       AND NOT "LBP_Axis08_W".E_PLCASp;
   END_REGION

   REGION Axis PLC mode (When NC Not in JOG Mode)
       IF #sAxisCNCMode
            AND #iPLCModeReq THEN
           #sAxisPLCMode := TRUE;
           #sAxisCNCMode := FALSE;
       END_IF;

       #sAllAxisPLCMode :=
           "LBP_Axis05_U1".E_PLCASp
       AND "LBP_Axis06_U2".E_PLCASp
       AND "LBP_Axis07_V".E_PLCASp
       AND "LBP_Axis08_W".E_PLCASp;
   END_REGION

   REGION Set axis feed rate
       #sU1ActFeedRate := "DB_AxisPosition".sAxis05_U1."$MA_MAX_AX_VELO";
       #sU2ActFeedRate := "DB_AxisPosition".sAxis06_U2."$MA_MAX_AX_VELO";
       #sVActFeedRate := "DB_AxisPosition".sAxis07_V."$MA_MAX_AX_VELO";
       IF (("DB_LoaderShuttle1".sIntLoadUnload.sCurrent_Step_NB = 100
           OR "DB_LoaderShuttle1".sIntLoadUnload.sCurrent_Step_NB = 110)
           AND "DB_AxisPosition".sAxis08_W."$AA_IM" <= "DB_AxisPosMachinePLC".Axis_W.Shuttle_1.Approach)

           OR (("DB_LoaderShuttle2".sIntLoadUnload.sCurrent_Step_NB = 100
           OR "DB_LoaderShuttle2".sIntLoadUnload.sCurrent_Step_NB = 110)
           AND "DB_AxisPosition".sAxis08_W."$AA_IM" <= "DB_AxisPosMachinePLC".Axis_W.Shuttle_2.Approach)

           OR (("DB_LoaderShuttle1".sIntLoadUnloadOP.sCurrent_Step_NB = 100
           OR "DB_LoaderShuttle1".sIntLoadUnloadOP.sCurrent_Step_NB = 110)
           AND "DB_AxisPosition".sAxis08_W."$AA_IM" <= "DB_AxisPosMachinePLC".Axis_W.Shuttle_1.Approach)

           OR (("DB_LoaderShuttle2".sIntLoadUnloadOP.sCurrent_Step_NB = 100
           OR "DB_LoaderShuttle2".sIntLoadUnloadOP.sCurrent_Step_NB = 110)
           AND "DB_AxisPosition".sAxis08_W."$AA_IM" <= "DB_AxisPosMachinePLC".Axis_W.Shuttle_2.Approach)

           OR (("DB_LoaderShuttle1".sIntLoadUnloadOP.sCurrent_Step_NB = 190
           OR "DB_LoaderShuttle1".sIntLoadUnloadOP.sCurrent_Step_NB = 200)
           AND "DB_AxisPosition".sAxis08_W."$AA_IM" <= "DB_AxisPosMachinePLC".Axis_W.Shuttle_1.Approach)

           OR (("DB_LoaderShuttle2".sIntLoadUnloadOP.sCurrent_Step_NB = 190
           OR "DB_LoaderShuttle2".sIntLoadUnloadOP.sCurrent_Step_NB = 200)
           AND "DB_AxisPosition".sAxis08_W."$AA_IM" <= "DB_AxisPosMachinePLC".Axis_W.Shuttle_2.Approach)

           OR(("DB_LoaderFixture".sFixtureLoading.sCurrent_Step_NB = 80
           OR "DB_LoaderFixture".sFixtureLoading.sCurrent_Step_NB = 85)
           AND "DB_AxisPosition".sAxis08_W."$AA_IM" <= "DB_AxisPosMachinePLC".Axis_W.Fixture.Approach)


       THEN
           #sWActFeedRate := "DB_AxisPosition".sAxis08_W."$MA_JOG_VELO";
       ELSE
           #sWActFeedRate := "DB_AxisPosition".sAxis08_W."$MA_MAX_AX_VELO";
       END_IF;
   END_REGION

   REGION Check axis drived by PLC
       // Axis U1
       #sU1DrivedByPLC := "LBP_Axis05_U1".E_RefSyn1
       AND #sAxisPLCMode
       AND NOT #sAxisCNCMode;

       // Axis U2
       #sU2DrivedByPLC := "LBP_Axis06_U2".E_RefSyn1
       AND #sAxisPLCMode
       AND NOT #sAxisCNCMode;

       // Axis V
       #sVDrivedByPLC := "LBP_Axis07_V".E_RefSyn1
       AND #sAxisPLCMode
       AND NOT #sAxisCNCMode;

       // Axis W
       #sWDrivedByPLC := "LBP_Axis08_W".E_RefSyn1
       AND #sAxisPLCMode
       AND NOT #sAxisCNCMode;
   END_REGION

   REGION Set axis PLC/CNC mode
       // Axis U1 (Always drived by PLC in Auto Mode)
       "LBP_Axis05_U1".A_NCASpStrobe := #sU1DrivedByPLC
       AND NOT "LBP_Axis05_U1".E_PLCASp
       OR NOT #sU1DrivedByPLC
       AND "LBP_Axis05_U1".E_PLCASp;

       "LBP_Axis05_U1".A_PLCASp := #sU1DrivedByPLC;

       // Axis U2 (Always drived by PLC in Auto Mode)
       "LBP_Axis06_U2".A_NCASpStrobe := #sU2DrivedByPLC
       AND NOT "LBP_Axis06_U2".E_PLCASp
       OR NOT #sU2DrivedByPLC
       AND "LBP_Axis06_U2".E_PLCASp;

       "LBP_Axis06_U2".A_PLCASp := #sU2DrivedByPLC;

       // Axis V (Always drived by PLC in Auto Mode)
       "LBP_Axis07_V".A_NCASpStrobe := #sVDrivedByPLC
       AND NOT "LBP_Axis07_V".E_PLCASp
       OR NOT #sVDrivedByPLC
       AND "LBP_Axis07_V".E_PLCASp;

       "LBP_Axis07_V".A_PLCASp := #sVDrivedByPLC;

       // Axis W (Always drived by PLC in Auto Mode)
       "LBP_Axis08_W".A_NCASpStrobe := #sWDrivedByPLC
       AND NOT "LBP_Axis08_W".E_PLCASp
       OR NOT #sWDrivedByPLC
       AND "LBP_Axis08_W".E_PLCASp;

       "LBP_Axis08_W".A_PLCASp := #sWDrivedByPLC;
   END_REGION

   REGION Delete distance to go
       // Axis U1
       "LBP_Axis05_U1".A_DelDTGSpReset := NOT #sU1StartMove
       AND "LBP_Axis05_U1".E_PLCASp
       OR "MCP1_In".reset
       OR "LBP_ModeGroup".E_REF;

       // Axis U2
       "LBP_Axis06_U2".A_DelDTGSpReset := NOT #sU2StartMove
       AND "LBP_Axis06_U2".E_PLCASp
       OR "MCP1_In".reset
       OR "LBP_ModeGroup".E_REF;

       // Axis V
       "LBP_Axis07_V".A_DelDTGSpReset := NOT #sVStartMove
       AND "LBP_Axis07_V".E_PLCASp
       OR "MCP1_In".reset
       OR "LBP_ModeGroup".E_REF;

       // Axis W
       "LBP_Axis08_W".A_DelDTGSpReset := NOT #sWStartMove
       AND "LBP_Axis08_W".E_PLCASp
       OR "MCP1_In".reset
       OR "LBP_ModeGroup".E_REF;
   END_REGION

   REGION Axis positioning
       // Axis U1
       "LBP_CtrlAxisSpindle"(Start := #sU1StartMove AND #sU1DrivedByPLC,
                             Stop := FALSE,
                             Funct := B#16#5,
                             Mode := B#16#0,
                             AxisNo := 5,
                             Pos := #sU1SetPos,
                             FRate := LREAL_TO_REAL(#sU1ActFeedRate),
                             InPos => #sU1InPos,
                             Error => #sU1MoveError,
                             State => #sU1MoveState);

       IF #sU1InPos
           OR "MCP1_In".reset
           OR #sU1MoveError THEN
           #sU1StartMove := FALSE;
       END_IF;

       IF #sU1MoveError THEN
           "LBP_AlarmMsgs".UserA[08].A70UUxx[08] := TRUE;
       END_IF;

       // Axis U2
       "LBP_CtrlAxisSpindle"(Start := #sU2StartMove AND #sU2DrivedByPLC,
                             Stop := FALSE,
                             Funct := B#16#5,
                             Mode := B#16#0,
                             AxisNo := 6,
                             Pos := #sU2SetPos,
                             FRate := LREAL_TO_REAL(#sU2ActFeedRate),
                             InPos => #sU2InPos,
                             Error => #sU2MoveError,
                             State => #sU2MoveState);
       IF #sU2MoveState <> 0 THEN
           "DB_WAF".U2States := #sU2MoveState;
       END_IF;

       IF #sU2InPos
           OR "MCP1_In".reset
           OR #sU2MoveError THEN
           #sU2StartMove := FALSE;
       END_IF;

       IF #sU2MoveError THEN
           "LBP_AlarmMsgs".UserA[08].A70UUxx[09] := TRUE;
       END_IF;

       // Axis V
       "LBP_CtrlAxisSpindle"(Start := #sVStartMove AND #sVDrivedByPLC,
                             Stop := FALSE,
                             Funct := B#16#5,
                             Mode := B#16#0,
                             AxisNo := 7,
                             Pos := #sVSetPos,
                             FRate := LREAL_TO_REAL(#sVActFeedRate),
                             InPos => #sVInPos,
                             Error => #sVMoveError,
                             State => #sVMoveState);

       IF #sVInPos
           OR "MCP1_In".reset
           OR #sVMoveError THEN
           #sVStartMove := FALSE;
       END_IF;

       IF #sVMoveError THEN
           "LBP_AlarmMsgs".UserA[08].A70UUxx[10] := TRUE;
       END_IF;

       // Axis W
       "LBP_CtrlAxisSpindle"(Start := #sWStartMove AND #sWDrivedByPLC,
                             Stop := FALSE,
                             Funct := B#16#5,
                             Mode := B#16#0,
                             AxisNo := 8,
                             Pos := #sWSetPos,
                             FRate := LREAL_TO_REAL(#sWActFeedRate),
                             InPos => #sWInPos,
                             Error => #sWMoveError,
                             State => #sWMoveState);

       IF #sWInPos
           OR "MCP1_In".reset
           OR #sWMoveError THEN
           #sWStartMove := FALSE;
       END_IF;

       IF #sWMoveError THEN
           "LBP_AlarmMsgs".UserA[08].A70UUxx[11] := TRUE;
       END_IF;
   END_REGION

   REGION Update Outputs
       #oU1InPos := #sU1InPos;
       #oU2InPos := #sU2InPos;
       #oVInPos  := #sVInPos;
       #oWInPos  := #sWInPos;
   END_REGION
END_FUNCTION_BLOCK

FUNCTION_BLOCK "FB_GestionSafetyGate"   // FB202, SCL
{ S7_Optimized_Access := 'TRUE' }
// stored: AutoNumber false, MemoryReserve 100, SetENOAutomatically false
   VAR
      sExtGate { S7_SetPoint := 'True'} : "FB_CmdCylinder";
      sIntGate { S7_SetPoint := 'True'} : "FB_CmdCylinder";
      sExtGateCloseCmd : Bool;
      sExtGateOpenCmd : Bool;
      sIntGateCloseCmd : Bool;
      sIntGateOpenCmd : Bool;
      sJOG_Cmd : Bool;
      sRT_RefCmd : R_TRIG;
      sFT_RefCmd : F_TRIG;
      sExtGateOpenReq : Bool;
      sIntGateOpenReq : Bool;
      sExtGateOpened : Bool;
      sExtGateClosed : Bool;
      sIntGateOpened : Bool;
      sIntGateClosed : Bool;
      sWaitCloseShutterBeforeOpen : Bool;
      sWaitOpenShutterAfterClose : Bool;
      sTimeoutOpenCloseGateTimer : TON_TIME;
      sRT_IntGateOpenbyHMI { S7_SetPoint := 'True'} : R_TRIG;
      sFT_IntGateOpenbyHMI { S7_SetPoint := 'True'} : F_TRIG;
      sRT_ExtGateOpenbyHMI { S7_SetPoint := 'True'} : R_TRIG;
      sFT_ExtGateOpenbyHMI { S7_SetPoint := 'True'} : F_TRIG;
      sRT_ExtGateClose { S7_SetPoint := 'True'} : R_TRIG;
      sRT_ExtGateOpen { S7_SetPoint := 'True'} : R_TRIG;
      sRT_IntGateClose { S7_SetPoint := 'True'} : R_TRIG;
      sRT_IntGateOpen { S7_SetPoint := 'True'} : R_TRIG;
      sInterlockExtGateClose { S7_SetPoint := 'True'} : Bool;
      sInterlockExtGateOpen { S7_SetPoint := 'True'} : Bool;
      sInterlockIntGateClose : Bool;
      sInterlockIntGateOpen : Bool;
   END_VAR
   VAR_TEMP
      tError : Int;
      tCloseExtGate : Bool;
      tOpenExtGate : Bool;
      tCloseIntGate : Bool;
      tOpenIntGate : Bool;
      tSasPosShuttle1 : Real;
      tSasPosShuttle2 : Real;
      tActPosShuttle1 : Real;
      tActPosShuttle2 : Real;
      tDeltaSasShuttle1 : Real;
      tDeltaSasShuttle2 : Real;
      tSynchroMode : Bool;
      tOpenAllGates : Bool;
      tCloseAllGates : Bool;
   END_VAR
   VAR CONSTANT
      TIMEOUT_OPEN_CLOSE_GATE_TIME : Time := T#3s;
   END_VAR
BEGIN
   REGION Description header 
       //==================================================================================
       // POSALUX Swiss SA / (C) Copyright 2025
       //----------------------------------------------------------------------------------
       // Title: Initialization of axis
       // Comment/Function: 
       // Author: Fabien WALDT
       // Engineering: TIA Portal v17
       //----------------------------------------------------------------------------------
       // Change log table:
       // Version  | Date     | Expert in charge | Changes applied
       // ---------|----------|------------------|-----------------------------------------
       // 00.00.01 | 20250509 | WFA              | First released version
       // =================================================================================
   END_REGION

   REGION Reference - Jog Command : Open/Close all Gates
       // Si mode Jog ET Demande reference OU Axe Shuttle selectionné, ouverture SAS Int et Ext
       #sRT_RefCmd(CLK := (("LBP_Chan1".A_Ref OR "MCP1_Out".LEDaxis5 OR "MCP1_Out".LEDaxis6) AND "LBP_ModeGroup".E_JOG)
                  OR "LBP_Chan1".MDyn[45]);     // M45: Open all Gates

       IF #sRT_RefCmd.Q THEN
           #sWaitCloseShutterBeforeOpen := TRUE;
       END_IF;

       IF #sRT_RefCmd.Q THEN
           #tCloseAllGates := FALSE;
       END_IF;

      // #tOpenAllGates := #Wait_close_Shutter_before_open AND ("DB_DataFromSafety".ShutterOpened OR NOT "DB_DataFromSafety".EmergencyStop); WFA A mettre en place quand shutter OK
       #tOpenAllGates := #sWaitCloseShutterBeforeOpen AND (true OR NOT "DB_DataFromSafety".EmergencyStop);

      IF #tOpenAllGates THEN
          #sWaitCloseShutterBeforeOpen := FALSE;
      END_IF;

       #sFT_RefCmd(CLK := (("LBP_Chan1".A_Ref OR "MCP1_Out".LEDaxis5 OR "MCP1_Out".LEDaxis6) AND "LBP_ModeGroup".E_JOG)
                  OR "LBP_Chan1".MDyn[44]);     // M44: Close all Gates

       IF #sFT_RefCmd.Q THEN
           #tCloseAllGates := TRUE;
       END_IF;

       IF #sFT_RefCmd.Q THEN
           #sWaitCloseShutterBeforeOpen := FALSE;
       END_IF;
   END_REGION

   REGION Close Shutter when all gates are open
       IF "LBP_Chan1".MDyn[45] THEN                // M45: Open all Gates
           "DB_DataToSafety".CloseShutter := TRUE;
       END_IF;

       IF "MCP1_In".reset
           OR "LBP_Chan1".MDyn[44] THEN           // M44: Close all Gates
           #sWaitOpenShutterAfterClose := TRUE;
       END_IF;

       IF #sWaitOpenShutterAfterClose AND (NOT "DB_DigitalInputs".sExternalGateLocked.sSWStatus OR NOT "DB_DigitalInputs".sInternalGateLocked.sSWStatus) THEN
           #sWaitOpenShutterAfterClose := FALSE;
           "DB_DataToSafety".CloseShutter := FALSE;
       END_IF;
   END_REGION

   REGION Time Out Gate
       #sTimeoutOpenCloseGateTimer(IN := NOT (("LBP_Chan1".A_Ref OR "MCP1_Out".LEDaxis5 OR "MCP1_Out".LEDaxis6) AND "LBP_ModeGroup".E_JOG) AND (NOT "DB_DigitalInputs".sExternalGateLocked.sSWStatus OR NOT "DB_DigitalInputs".sInternalGateLocked.sSWStatus),
                                   PT := #TIMEOUT_OPEN_CLOSE_GATE_TIME);

       IF #sTimeoutOpenCloseGateTimer.Q THEN
           "LBP_AlarmMsgs".UserA[2].A70UUxx[18]:= TRUE;     // Msg: "700218 - Time out doors SAS int/ext"
       END_IF;
   END_REGION

   REGION Gates management by HMI
       IF "LBP_ModeGroup".E_JOG
           AND NOT "LBP_Chan1".A_Ref
           AND NOT "MCP1_Out".LEDaxis5
           AND NOT "MCP1_Out".LEDaxis6 THEN
           #sRT_IntGateOpenbyHMI(CLK := "DB_HMICmd".IntGateOpenReq,
                                 Q => "DB_HMICmd".IntGateOpenCmd);

           #sFT_IntGateOpenbyHMI(CLK := "DB_HMICmd".IntGateOpenReq,
                                 Q => "DB_HMICmd".IntGateCloseCmd);

           #sRT_ExtGateOpenbyHMI(CLK := "DB_HMICmd".ExtGateOpenReq,
                                 Q => "DB_HMICmd".ExtGateOpenCmd);

           #sFT_ExtGateOpenbyHMI(CLK := "DB_HMICmd".ExtGateOpenReq,
                                 Q => "DB_HMICmd".ExtGateCloseCmd);
       END_IF;
   END_REGION

   REGION Syncro Mode
       #tSynchroMode := "DB_LoaderShuttle1".sMain.sInterface.SequenceRun
       AND "DB_LoaderShuttle2".sMain.sInterface.SequenceRun
       AND (("DB_LoaderShuttle1".sShuttleInt.oExtGateOpenReq AND "DB_LoaderShuttle2".sShuttlePosSas)
         OR ("DB_LoaderShuttle1".sShuttleInt.oIntGateOpenReq AND "DB_LoaderShuttle2".sShuttlePosInt)
         OR ("DB_LoaderShuttle1".sShuttleExt.oExtGateOpenReq AND "DB_LoaderShuttle2".sShuttlePosExt)
         OR ("DB_LoaderShuttle1".sShuttleExt.oIntGateOpenReq AND "DB_LoaderShuttle2".sShuttlePosSas)
         OR ("DB_LoaderShuttle2".sShuttleInt.oExtGateOpenReq AND "DB_LoaderShuttle1".sShuttlePosSas)
         OR ("DB_LoaderShuttle2".sShuttleInt.oIntGateOpenReq AND "DB_LoaderShuttle1".sShuttlePosInt)
         OR ("DB_LoaderShuttle2".sShuttleExt.oExtGateOpenReq AND "DB_LoaderShuttle1".sShuttlePosExt)
         OR ("DB_LoaderShuttle2".sShuttleExt.oIntGateOpenReq AND "DB_LoaderShuttle1".sShuttlePosSas));
   END_REGION

   REGION Gates management by M Codes - PLC Sequence
       IF #tCloseAllGates THEN
           #sExtGateOpenReq := FALSE;
           #sIntGateOpenReq := FALSE;
       END_IF;

       // External Gate
       IF "LBP_Chan1".MDyn[46]                         // M46: Closing External Gate (Not in ISO Code)
           OR "DB_LoaderShuttle1".oExtGateCloseReq     // Closure External Gate request from Shuttle 1
           OR "DB_LoaderShuttle2".oExtGateCloseReq     // Closure External Gate request from Shuttle 2
           OR "DB_HMICmd".ExtGateCloseCmd THEN         // Closure External Gate request from HMI
               #sExtGateOpenReq := FALSE;
       END_IF;

       IF "LBP_Chan1".MDyn[47]                                                                                                                            // M47: Opening External Gate (Not in ISO Code)
           OR (("DB_LoaderShuttle1".oExtGateOpenReq OR "DB_LoaderShuttle2".oExtGateOpenReq) AND NOT "DB_LoaderMain".sSynchroMode AND NOT #tSynchroMode)   // Opening External Gate request from Shuttle 1 or 2 (Only one Shuttle sequence is running)
           OR (("DB_LoaderShuttle1".oExtGateOpenReq AND "DB_LoaderShuttle2".oExtGateOpenReq) AND ("DB_LoaderMain".sSynchroMode OR #tSynchroMode))         // Opening External Gate request from Shuttle 1 and 2 (both Shuttle sequence are running)
           OR "DB_HMICmd".ExtGateOpenCmd                                                                                                                  // Opening External Gate request from HMI
           OR (("LBP_Chan1".A_Ref OR "MCP1_Out".LEDaxis5 OR "MCP1_Out".LEDaxis6) AND "LBP_ModeGroup".E_JOG) THEN                                          // Opening External Gate request from Mode Group
               #sExtGateOpenReq := TRUE;
       END_IF;

       #sRT_ExtGateClose(CLK:=NOT  #sExtGateOpenReq AND NOT #sInterlockExtGateClose,
                             Q=> #tCloseExtGate);

       #sRT_ExtGateOpen(CLK := #sExtGateOpenReq AND NOT #sInterlockExtGateOpen,
                            Q => #tOpenExtGate);

        // Internal Gate
       IF "LBP_Chan1".MDyn[48]                         // M48: Closing Internal Gate (Not in ISO Code)
           OR "DB_LoaderShuttle1".oIntGateCloseReq     // Closure Internal Gate request from Shuttle 1
           OR "DB_LoaderShuttle2".oIntGateCloseReq     // Closure Internal Gate request from Shuttle 2
           OR "DB_HMICmd".IntGateCloseCmd THEN         // Closure External Gate request from HMI
               #sIntGateOpenReq := FALSE;
       END_IF;

       IF "LBP_Chan1".MDyn[49]                                                                                                                            // M49: Opening Internal Gate (Not in ISO Code)
           OR (("DB_LoaderShuttle1".oIntGateOpenReq OR "DB_LoaderShuttle2".oIntGateOpenReq) AND NOT "DB_LoaderMain".sSynchroMode AND NOT #tSynchroMode)   // Opening Internal Gate request from Shuttle 1 or 2 (Only one Shuttle sequence is running)
           OR (("DB_LoaderShuttle1".oIntGateOpenReq AND "DB_LoaderShuttle2".oIntGateOpenReq) AND ("DB_LoaderMain".sSynchroMode OR #tSynchroMode))         // Opening Internal Gate request from Shuttle 1 and 2 (both Shuttle sequence are running)
           OR "DB_HMICmd".IntGateOpenCmd                                                                                                                  // Opening External Gate request from HMI
           OR (("LBP_Chan1".A_Ref OR "MCP1_Out".LEDaxis5 OR "MCP1_Out".LEDaxis6) AND "LBP_ModeGroup".E_JOG) THEN                                          // Opening External Gate request from Mode Group
           #sIntGateOpenReq := TRUE;
       END_IF;

       #sRT_IntGateClose(CLK := NOT #sIntGateOpenReq AND NOT #sInterlockIntGateClose,
                          Q => #tCloseIntGate);

        #sRT_IntGateOpen(CLK := #sIntGateOpenReq AND NOT #sInterlockIntGateOpen,
                          Q => #tOpenIntGate);
    END_REGION

    REGION Interlocks
        #sInterlockExtGateOpen := NOT #sIntGateClosed OR #sIntGateOpenReq;
        #sInterlockIntGateOpen := NOT #sExtGateClosed OR #sExtGateOpenReq;

        #sInterlockExtGateClose := ("DB_AxisPosition".sAxis05_U1."$AA_IM" >= "DB_AxisPosMachinePLC".Axis_U1.ExtGateExt
        AND "DB_AxisPosition".sAxis05_U1."$AA_IM" <= "DB_AxisPosMachinePLC".Axis_U1.IntGateExt)
        OR ("DB_AxisPosition".sAxis06_U2."$AA_IM" >= "DB_AxisPosMachinePLC".Axis_U2.ExtGateExt
        AND "DB_AxisPosition".sAxis06_U2."$AA_IM" <= "DB_AxisPosMachinePLC".Axis_U2.IntGateExt);

        #sInterlockIntGateClose := ("DB_AxisPosition".sAxis05_U1."$AA_IM" >= "DB_AxisPosMachinePLC".Axis_U1.ExtGateInt
        AND "DB_AxisPosition".sAxis05_U1."$AA_IM" <= "DB_AxisPosMachinePLC".Axis_U1.IntGateInt)
        OR ("DB_AxisPosition".sAxis06_U2."$AA_IM" >= "DB_AxisPosMachinePLC".Axis_U2.ExtGateInt
        AND "DB_AxisPosition".sAxis06_U2."$AA_IM" <= "DB_AxisPosMachinePLC".Axis_U2.IntGateInt);
    END_REGION

    REGION External Gate Command
        #sExtGateCloseCmd := (#tCloseAllGates OR #tCloseExtGate) AND NOT #sInterlockExtGateClose;
        #sExtGateOpenCmd := #tOpenAllGates OR (#tOpenExtGate AND NOT #sInterlockExtGateOpen);
    END_REGION

    REGION Internal Gate Command
        #sIntGateCloseCmd := (#tCloseAllGates OR #tCloseIntGate) AND NOT #sInterlockIntGateClose;
        #sIntGateOpenCmd := #tOpenAllGates OR (#tOpenIntGate AND NOT #sInterlockIntGateOpen);
    END_REGION 

    REGION External Gate
        #sExtGate(iEMinus := "DB_DigitalInputs".sExternalGateLocked.sSWStatus,
                  iEPlus := "DB_DigitalInputs".sExternalGateOpened.sSWStatus,
                  iMinusCmd := #sExtGateCloseCmd,
                  iPlusCmd := #sExtGateOpenCmd,
                  iJOGCmd := #sJOG_Cmd,
                  iMonitorTime := T#8s,
                  oErrorCode => #tError,
                  ioQMinus := "DB_DigitalOutputs".sExternalGateClosing.sSWStatus,
                  ioQPlus := "DB_DigitalOutputs".sExternalGateOpening.sSWStatus);

        CASE #tError OF
            1:
                "LBP_AlarmMsgs".UserA[2].A70UUxx[21] := TRUE;  // Msg: "700221 - Time out door ext. SAS closing"
            2:
                "LBP_AlarmMsgs".UserA[2].A70UUxx[19] := TRUE;  // Msg: "700219 - Time out door ext. SAS opening"
        END_CASE;
    END_REGION ;

    REGION Internal Gate
        #sIntGate(iEMinus:= "DB_DigitalInputs".sInternalGateLocked.sSWStatus,
                  iEPlus:=  "DB_DigitalInputs".sInternalGateOpened.sSWStatus,
                  iMinusCmd:=#sIntGateCloseCmd,
                  iPlusCmd:=#sIntGateOpenCmd,
                  iJOGCmd:=#sJOG_Cmd,
                  iMonitorTime:=T#8s,
                  oErrorCode=>#tError,
                  ioQMinus:="DB_DigitalOutputs".sInternalGateClosing.sSWStatus,
                  ioQPlus:="DB_DigitalOutputs".sInternalGateOpening.sSWStatus);

        CASE #tError OF
            1:
               "LBP_AlarmMsgs".UserA[2].A70UUxx[22] := TRUE;  // Msg: "700222 - Time out door int. SAS closing" (WFA à corriger)
            2:
               "LBP_AlarmMsgs".UserA[2].A70UUxx[20] := TRUE;  // Msg: "700220 - Time out door int. SAS opening" (WFA à corriger)
        END_CASE;
    END_REGION ;

    REGION Gates Status 
        // External Gate Closed
        #sExtGateClosed := "DB_DigitalInputs".sExternalGateLocked.sSWStatus
        AND NOT "DB_DigitalInputs".sExternalGateOpened.sSWStatus;

        // External Gate Open
        #sExtGateOpened := NOT "DB_DigitalInputs".sExternalGateLocked.sSWStatus
        AND "DB_DigitalInputs".sExternalGateOpened.sSWStatus;

        // Internal Gate Closed
        #sIntGateClosed := "DB_DigitalInputs".sInternalGateLocked.sSWStatus
        AND NOT "DB_DigitalInputs".sInternalGateOpened.sSWStatus;

        // Internal Gate Open
        #sIntGateOpened := NOT "DB_DigitalInputs".sInternalGateLocked.sSWStatus
        AND "DB_DigitalInputs".sInternalGateOpened.sSWStatus;
    END_REGION ;
END_FUNCTION_BLOCK

FUNCTION_BLOCK "FB_CmdCylinder"   // FB44, SCL
{ S7_Optimized_Access := 'TRUE' }
// stored: AutoNumber false, MemoryReserve 100, SetENOAutomatically false
   VAR_INPUT
      iEMinus { ExternalAccessible := 'False'; ExternalVisible := 'False'; ExternalWritable := 'False'} : Bool;
      iEPlus { ExternalAccessible := 'False'; ExternalVisible := 'False'; ExternalWritable := 'False'} : Bool;
      iMinusCmd { ExternalAccessible := 'False'; ExternalVisible := 'False'; ExternalWritable := 'False'} : Bool;
      iPlusCmd { ExternalAccessible := 'False'; ExternalVisible := 'False'; ExternalWritable := 'False'} : Bool;
      iJOGCmd { ExternalAccessible := 'False'; ExternalVisible := 'False'; ExternalWritable := 'False'} : Bool;
      iMonitorTime : Time;
   END_VAR
   VAR_OUTPUT
      oMinusPos { ExternalAccessible := 'False'; ExternalVisible := 'False'; ExternalWritable := 'False'} : Bool;
      oMiddlePos { ExternalAccessible := 'False'; ExternalVisible := 'False'; ExternalWritable := 'False'} : Bool;
      oPlusPos { ExternalAccessible := 'False'; ExternalVisible := 'False'; ExternalWritable := 'False'} : Bool;
      oErrorCode { ExternalAccessible := 'False'; ExternalVisible := 'False'; ExternalWritable := 'False'} : Int;
   END_VAR
   VAR_IN_OUT
      ioQMinus { ExternalAccessible := 'False'; ExternalVisible := 'False'; ExternalWritable := 'False'} : Bool;
      ioQPlus { ExternalAccessible := 'False'; ExternalVisible := 'False'; ExternalWritable := 'False'} : Bool;
   END_VAR
   VAR
      sRT_NoCmd : R_TRIG;
      sMonitorTimer { S7_SetPoint := 'True'} : TON_TIME;
   END_VAR
BEGIN
   REGION Description header 
       //==================================================================================
       // POSALUX Swiss SA / (C) Copyright 2025
       //----------------------------------------------------------------------------------
       // Title: FB_CmdCylinder
       // Comment/Function: Cylinder management with 2 outputs (Cmd) and two inputs (Pos)
       //                   Movements and positions are monitored:
       //                      Error Code 0: No Error
       //                      Error Code 1: Error Timeout Command Plus
       //                      Error Code 2: Error Timeout Command Minus
       //                      Error Code 3: Error Timeout Position OFF   
       //                      Error Code 4: Error Timeout Position ON             
       // Author: Fabien WALDT
       // Engineering: TIA Portal v17
       //----------------------------------------------------------------------------------
       // Change log table:
       // Version  | Date     | Expert in charge | Changes applied
       // ---------|----------|------------------|-----------------------------------------
       // 00.00.01 | 20250501 | WFA              | First released version
       // =================================================================================
   END_REGION

   REGION Init
       // No command : both plus and minus are set. (WFA ??)
       #sRT_NoCmd(CLK:=NOT #ioQMinus AND NOT #ioQPlus);
       IF #sRT_NoCmd.Q THEN
           #ioQMinus := TRUE;
           #ioQPlus := TRUE;
           RETURN;
       END_IF;
   END_REGION

   REGION Plus / Minus Commands
       // Minus Command
       IF #iMinusCmd THEN
           #ioQPlus := FALSE;
           #ioQMinus := TRUE;
       END_IF;

       // Plus Command
       IF #iPlusCmd THEN
           #ioQMinus := FALSE;
           #ioQPlus := TRUE;
       END_IF;

       // JOG stop on the way : both plus and minus are set. (WFA ??)
       IF #iJOGCmd AND NOT #iMinusCmd AND NOT #iPlusCmd THEN
           #ioQMinus := TRUE;
           #ioQPlus := TRUE;
       END_IF;
   END_REGION

   REGION Positions
       #oMinusPos := #iEMinus AND NOT #iEPlus;
       #oMiddlePos := NOT #iEMinus AND NOT #iEPlus;
       #oPlusPos := #iEPlus AND NOT #iEMinus;
   END_REGION

   REGION Monitoring Timer
       #sMonitorTimer(IN:=(#iMinusCmd AND NOT #oMinusPos) OR
                      (#iPlusCmd AND NOT #oPlusPos) OR
                      (NOT #oMinusPos AND NOT #oPlusPos) OR
                      (#iEMinus AND #iEPlus),
                      PT:=#iMonitorTime);
   END_REGION

   REGION Error Codes
       #oErrorCode := 0;           // Code 0: No Error
       IF #iPlusCmd AND #sMonitorTimer.Q THEN
           #oErrorCode := 1;       // Code 1: Error Timeout Command Plus
       ELSIF #iMinusCmd AND #sMonitorTimer.Q THEN
           #oErrorCode := 2;       // Code 2: Error Timeout Command Minus
       ELSIF NOT #oMinusPos AND NOT #oPlusPos AND #sMonitorTimer.Q THEN
           #oErrorCode := 3;       // Code 3: Error Timeout Position OFF   
       ELSIF #iEMinus AND #iEPlus AND #sMonitorTimer.Q THEN
           #oErrorCode := 4;       // Code 4: Error Timeout Position ON       
       END_IF;
   END_REGION
END_FUNCTION_BLOCK

FUNCTION_BLOCK "FB_GestionGripper"   // FB43, SCL
{ S7_Optimized_Access := 'TRUE' }
// stored: MemoryReserve 100, SetENOAutomatically false
   VAR
      sLoadGripperCloseReq : Bool;
      sUnloadGripperCloseReq : Bool;
      sLoadShift : Bool;
      sUnLoadShift : Bool;
      sLoadPartLost : Bool;
      sUnLoadPartLost : Bool;
      sLoadClose : Bool;
      sUnLoadClose : Bool;
      sUndrilledGripper : "FB_Gripper";
      sDrilledGripper : "FB_Gripper";
      sLoadCloseWithPart : Bool;
      sUnLoadCloseWithPart : Bool;
      sLoadOpen : Bool;
      sUnLoadOpen : Bool;
      sFT_ModeJog : F_TRIG;
      sBlowingTimerCmdHMI : TP_TIME;
      sRT_BlowingCmdHMI { S7_SetPoint := 'True'} : R_TRIG;
      sBlowingISO { S7_SetPoint := 'True'} : Bool;
      sGripperStatus : Struct
         Available : Bool;
         DrivedByShuttle1 : Bool;
         DrivedByShuttle2 : Bool;
         DrivedByFixture : Bool;
      END_STRUCT;
      sGripperReq : Struct
         ByShuttle1 : Bool;
         ByShuttle2 : Bool;
         ByFixture : Bool;
      END_STRUCT;
      sUndrilledGripperErrorCode : Int;
      sDrilledGripperErrorCode : Int;
   END_VAR
   VAR_TEMP
      tLoadInCycle : Bool;
      tUnloadInCycle : Bool;
   END_VAR
BEGIN
   REGION Description header 
       //==================================================================================
       // POSALUX Swiss SA / (C) Copyright 2025
       //----------------------------------------------------------------------------------
       // Title: 
       // Comment/Function: 
       // Author: Fabien WALDT
       // Engineering: TIA Portal v17
       //----------------------------------------------------------------------------------
       // Change log table:
       // Version  | Date     | Expert in charge | Changes applied
       // ---------|----------|------------------|-----------------------------------------
       // 00.00.01 | 20250506 | WFA              | First released version
       // =================================================================================
   END_REGION

   REGION Key[4] and Key[5] Management
       // Key[4] : Activating of loading/unloading undrilled part
       // Key[5] : Activation of loading/unloading drilled part

       // Key[4] and Key[5] enabled in Jog Mode
       "DB_McpKeyboardSignals".sK4_GripperUndrilledPart.sKeyDisable := NOT "LBP_ModeGroup".E_JOG OR "DB_GestionWorkingModes".sMCP_KxxKeysDisable;
       "DB_HmiKeyboardSignals".sK4a_GripperUndrilledPartClose.sKeyDisable := NOT "LBP_ModeGroup".E_JOG;
       "DB_HmiKeyboardSignals".sK4b_GripperUndrilledPartOpen.sKeyDisable := NOT "LBP_ModeGroup".E_JOG;
       "DB_McpKeyboardSignals".sK5_GripperDrilledPart.sKeyDisable   := NOT "LBP_ModeGroup".E_JOG OR "DB_GestionWorkingModes".sMCP_KxxKeysDisable;
       "DB_HmiKeyboardSignals".sK5a_GripperDrilledPartClose.sKeyDisable   := NOT "LBP_ModeGroup".E_JOG;
   END_REGION

   REGION Load Gripper Command (Undrilled Part)
       // Load Gripper Close Command
       IF "LBP_Chan1".MDyn[80]     // M80 : Close/vaccum loader load (Undrilled Part)
           OR "DB_LoaderShuttle1".oLoadGripperCloseReq
           OR "DB_LoaderShuttle2".oLoadGripperCloseReq
           OR ("LBP_ModeGroup".E_JOG AND "DB_McpKeyboardSignals".sK4_GripperUndrilledPart.sKeySWTogglePositiveFront) 
           OR ("LBP_ModeGroup".E_JOG AND "DB_HmiKeyboardSignals".sK4a_GripperUndrilledPartClose.sKeySWPositiveFront) THEN
           #sLoadGripperCloseReq := TRUE;
       END_IF;

       // Load Gripper Open Command
        IF "LBP_Chan1".MDyn[81]     // M81 : Open/blowing loader load (Undrilled Part)
            OR "DB_LoaderFixture".oLoadGripperOpenReq
            OR ("LBP_ModeGroup".E_JOG AND "DB_McpKeyboardSignals".sK4_GripperUndrilledPart.sKeySWToggleNegativeFront) 
           OR ("LBP_ModeGroup".E_JOG AND "DB_HmiKeyboardSignals".sK4b_GripperUndrilledPartOpen.sKeySWPositiveFront) THEN
           #sLoadGripperCloseReq := FALSE;
        END_IF;
       "DB_McpKeyboardSignals".sK4_GripperUndrilledPart.sKeySWToggleStatus := #sLoadGripperCloseReq;
      // "DB_HmiKeyboardSignals".sK4a_GripperUndrilledPartClose.sKeySWToggleStatus := #sLoadGripperCloseReq;
   END_REGION

   REGION Unload Gripper Command (Drilled Part)  
       // Unload Gripper Close Command
       IF "LBP_Chan1".MDyn[82]     // M82 : Close/vaccum loader unload (Drilled Part)
           OR "DB_LoaderFixture".oUnloadGripperCloseReq
           OR ("LBP_ModeGroup".E_JOG AND "DB_McpKeyboardSignals".sK5_GripperDrilledPart.sKeySWTogglePositiveFront)
           OR ("LBP_ModeGroup".E_JOG AND "DB_HmiKeyboardSignals".sK5a_GripperDrilledPartClose.sKeySWPositiveFront) THEN
           #sUnloadGripperCloseReq := TRUE;
       END_IF;

       // Unload Gripper Open Command
        IF "LBP_Chan1".MDyn[83]     // M83 : Open/blowing loader unload (Drilled Part)
           // OR #sLoadPartLost
           OR "DB_LoaderShuttle1".oUnloadGripperOpenReq
            OR "DB_LoaderShuttle2".oUnloadGripperOpenReq
         OR ("LBP_ModeGroup".E_JOG AND "DB_McpKeyboardSignals".sK5_GripperDrilledPart.sKeySWToggleNegativeFront)
          OR ("LBP_ModeGroup".E_JOG AND "DB_HmiKeyboardSignals".sK5b_GripperDrilledPartOpen.sKeySWTogglePositiveFront) THEN
            #sUnloadGripperCloseReq := FALSE;
       END_IF;
       "DB_McpKeyboardSignals".sK5_GripperDrilledPart.sKeySWToggleStatus := #sUnloadGripperCloseReq;
       "DB_HmiKeyboardSignals".sK5a_GripperDrilledPartClose.sKeySWToggleStatus := #sUnloadGripperCloseReq;
   END_REGION

   REGION Keys - LED Management
       // KEY - LED [4]: Loading (Undrilled part)
       "DB_McpKeyboardSignals".sK4_GripperUndrilledPart.sKeySWStatus :=
       #sLoadGripperCloseReq
       AND "DB_DecodChannels".sChan1IsDisplayed;

       "DB_HmiKeyboardSignals".sK4a_GripperUndrilledPartClose.sKeySWStatus :=
       #sLoadGripperCloseReq
       AND "DB_DecodChannels".sChan1IsDisplayed;

       "DB_HmiKeyboardSignals".sK4b_GripperUndrilledPartOpen.sKeySWStatus :=
       NOT #sLoadGripperCloseReq
       AND "DB_DecodChannels".sChan1IsDisplayed;

       "DB_McpKeyboardSignals".sK4_GripperUndrilledPart.sLedSWStatus := "DB_McpKeyboardSignals".sK4_GripperUndrilledPart.sKeySWStatus;
       "DB_HmiKeyboardSignals".sK4a_GripperUndrilledPartClose.sLedSWStatus := "DB_HmiKeyboardSignals".sK4a_GripperUndrilledPartClose.sKeySWStatus;
       "DB_HmiKeyboardSignals".sK4b_GripperUndrilledPartOpen.sLedSWStatus := "DB_HmiKeyboardSignals".sK4b_GripperUndrilledPartOpen.sKeySWStatus;

       // KEY - LED [5]: Unloading (Drilled part)
       "DB_McpKeyboardSignals".sK5_GripperDrilledPart.sKeySWStatus :=
       #sUnloadGripperCloseReq
       AND "DB_DecodChannels".sChan1IsDisplayed;

       "DB_HmiKeyboardSignals".sK5a_GripperDrilledPartClose.sKeySWStatus :=
       #sUnloadGripperCloseReq
       AND "DB_DecodChannels".sChan1IsDisplayed;

       "DB_HmiKeyboardSignals".sK5b_GripperDrilledPartOpen.sKeySWStatus :=
       NOT #sUnloadGripperCloseReq
       AND "DB_DecodChannels".sChan1IsDisplayed;

